C01801=1137.376,317.173,-76.633,-176.855,8.942,148.875
C01802=1137.380,316.925,-76.599,-176.858,8.938,148.874
C01803=1137.384,316.677,-76.568,-176.860,8.935,148.874
C01804=1137.388,316.429,-76.534,-176.863,8.931,148.874
C01805=1137.392,316.181,-76.503,-176.866,8.928,148.874
C01806=1137.396,315.933,-76.470,-176.869,8.923,148.874
C01807=1137.400,315.685,-76.439,-176.871,8.920,148.873
C01808=1137.405,315.438,-76.406,-176.874,8.916,148.873
C01809=1137.408,315.190,-76.374,-176.876,8.913,148.873
C01810=1137.413,314.941,-76.341,-176.879,8.909,148.873
C01811=1137.416,314.694,-76.309,-176.882,8.906,148.873
C01812=1137.420,314.447,-76.277,-176.885,8.902,148.873
C01813=1137.425,314.198,-76.245,-176.887,8.899,148.872
C01814=1137.429,313.950,-76.213,-176.890,8.894,148.872
C01815=1137.433,313.702,-76.180,-176.893,8.891,148.872
C01816=1137.437,313.424,-76.145,-176.896,8.887,148.872
C01817=1137.442,313.146,-76.109,-176.898,8.883,148.872
C01818=1137.447,312.868,-76.072,-176.901,8.879,148.871
C01819=1137.451,312.590,-76.036,-176.905,8.874,148.871
C01820=1137.456,312.342,-76.004,-176.907,8.871,148.871
C01821=1137.460,312.095,-75.973,-176.910,8.868,148.871
C01822=1137.464,311.847,-75.941,-176.913,8.864,148.870
C01823=1137.468,311.598,-75.908,-176.915,8.860,148.870
C01824=1137.472,311.350,-75.876,-176.918,8.856,148.870
C01825=1137.476,311.103,-75.845,-176.920,8.853,148.870
C01826=1137.481,310.855,-75.813,-176.924,8.849,148.870
C01827=1137.484,310.606,-75.781,-176.926,8.846,148.870
C01828=1137.489,310.359,-75.749,-176.929,8.842,148.869
C01829=1137.493,310.111,-75.717,-176.931,8.839,148.869
C01830=1137.497,309.863,-75.685,-176.934,8.835,148.869
C01831=1137.501,309.615,-75.653,-176.936,8.831,148.869
C01832=1137.505,309.367,-75.622,-176.939,8.827,148.869
C01833=1137.509,309.119,-75.589,-176.942,8.824,148.868
C01834=1137.513,308.872,-75.558,-176.945,8.820,148.868
C01835=1137.517,308.624,-75.526,-176.947,8.817,148.868
C01836=1137.521,308.376,-75.494,-176.950,8.814,148.868
C01837=1137.526,308.128,-75.462,-176.953,8.810,148.868
C01838=1137.530,307.879,-75.431,-176.955,8.806,148.868
C01839=1137.534,307.631,-75.399,-176.958,8.802,148.868
C01840=1137.538,307.384,-75.367,-176.960,8.799,148.867
C01841=1137.542,307.136,-75.336,-176.964,8.795,148.867
C01842=1137.547,306.888,-75.304,-176.966,8.792,148.867
C01843=1137.551,306.640,-75.272,-176.969,8.788,148.867
C01844=1137.554,306.392,-75.241,-176.971,8.785,148.867
C01845=1137.559,306.144,-75.209,-176.974,8.782,148.867
C01846=1137.562,305.896,-75.177,-176.977,8.777,148.866
C01847=1137.567,305.648,-75.146,-176.979,8.775,148.866
C01848=1137.571,305.400,-75.115,-176.982,8.770,148.866
C01849=1137.575,305.152,-75.082,-176.985,8.767,148.866
C01850=1137.580,304.904,-75.051,-176.988,8.763,148.866
C01851=1137.584,304.656,-75.020,-176.990,8.760,148.866
C01852=1137.588,304.409,-74.988,-176.993,8.757,148.866
C01853=1137.592,304.160,-74.957,-176.996,8.753,148.865
C01854=1137.596,303.913,-74.925,-176.998,8.750,148.865
C01855=1137.600,303.664,-74.894,-177.001,8.746,148.865
C01856=1137.604,303.417,-74.863,-177.003,8.742,148.865
C01857=1137.608,303.168,-74.831,-177.006,8.739,148.865
C01858=1137.613,302.921,-74.800,-177.009,8.735,148.865
C01859=1137.617,302.672,-74.768,-177.011,8.732,148.865
C01860=1137.621,302.425,-74.738,-177.014,8.728,148.864
C01861=1137.625,302.176,-74.706,-177.017,8.725,148.864
C01862=1137.629,301.929,-74.675,-177.019,8.722,148.864
C01863=1137.633,301.680,-74.643,-177.022,8.718,148.864
C01864=1137.638,301.433,-74.612,-177.025,8.714,148.864
C01865=1137.641,301.184,-74.581,-177.028,8.711,148.864
C01866=1137.646,300.937,-74.550,-177.030,8.707,148.864
C01867=1137.650,300.688,-74.519,-177.033,8.704,148.863
C01868=1137.654,300.441,-74.487,-177.036,8.700,148.863
C01869=1137.658,300.192,-74.456,-177.038,8.697,148.863
C01870=1137.663,299.945,-74.425,-177.041,8.693,148.863
C01871=1137.667,299.696,-74.393,-177.044,8.690,148.863
C01872=1137.671,299.448,-74.363,-177.047,8.687,148.863
C01873=1137.676,299.201,-74.331,-177.049,8.683,148.863
C01874=1137.680,298.952,-74.300,-177.052,8.680,148.863
C01875=1137.684,298.704,-74.269,-177.055,8.676,148.862
C01876=1137.687,298.456,-74.238,-177.057,8.673,148.862
C01877=1137.692,298.208,-74.207,-177.060,8.669,148.862
C01878=1137.696,297.960,-74.176,-177.063,8.665,148.862
C01879=1137.700,297.712,-74.145,-177.066,8.662,148.862
C01880=1137.705,297.464,-74.114,-177.068,8.659,148.862
C01881=1137.709,297.216,-74.083,-177.071,8.655,148.862
C01882=1137.713,296.968,-74.053,-177.074,8.652,148.862
C01883=1137.717,296.719,-74.022,-177.077,8.648,148.861
C01884=1137.721,296.471,-73.991,-177.079,8.645,148.861
C01885=1137.726,296.224,-73.959,-177.082,8.642,148.861
C01886=1137.730,295.975,-73.928,-177.085,8.638,148.861
C01887=1137.734,295.728,-73.898,-177.087,8.635,148.861
C01888=1137.738,295.480,-73.867,-177.090,8.632,148.861
C01889=1137.742,295.231,-73.836,-177.093,8.628,148.861
C01890=1137.746,294.983,-73.806,-177.095,8.624,148.861
C01891=1137.751,294.736,-73.775,-177.098,8.621,148.861
C01892=1137.755,294.487,-73.744,-177.101,8.617,148.860
C01893=1137.759,294.239,-73.713,-177.103,8.614,148.860
C01894=1137.763,293.991,-73.683,-177.106,8.610,148.860
C01895=1137.767,293.743,-73.652,-177.109,8.607,148.860
C01896=1137.772,293.495,-73.621,-177.111,8.604,148.860
C01897=1137.776,293.247,-73.591,-177.115,8.600,148.860
C01898=1137.780,292.998,-73.560,-177.117,8.597,148.860
C01899=1137.784,292.750,-73.529,-177.120,8.594,148.860
C01900=1137.788,292.503,-73.499,-177.123,8.590,148.860
C01901=1137.792,292.254,-73.468,-177.125,8.587,148.859
C01902=1137.796,292.006,-73.438,-177.128,8.584,148.859
C01903=1137.801,291.758,-73.407,-177.131,8.580,148.859
C01904=1137.805,291.511,-73.376,-177.133,8.577,148.859
C01905=1137.809,291.262,-73.346,-177.136,8.573,148.859
C01906=1137.813,291.014,-73.315,-177.139,8.569,148.859
C01907=1137.817,290.766,-73.285,-177.141,8.566,148.859
C01908=1137.822,290.518,-73.255,-177.144,8.563,148.859
C01909=1137.826,290.269,-73.223,-177.147,8.559,148.859
C01910=1137.830,290.022,-73.193,-177.150,8.556,148.859
C01911=1137.834,289.774,-73.163,-177.152,8.553,148.859
C01912=1137.839,289.525,-73.133,-177.155,8.550,148.859
C01913=1137.843,289.277,-73.102,-177.158,8.546,148.858
C01914=1137.846,289.029,-73.072,-177.160,8.543,148.858
C01915=1137.851,288.781,-73.041,-177.163,8.540,148.858
C01916=1137.855,288.533,-73.012,-177.166,8.536,148.858
C01917=1137.860,288.285,-72.981,-177.168,8.533,148.858
C01918=1137.863,288.037,-72.950,-177.171,8.530,148.858
C01919=1137.868,287.788,-72.920,-177.174,8.526,148.858
C01920=1137.873,287.513,-72.887,-177.177,8.523,148.858
C01921=1137.878,287.237,-72.853,-177.180,8.519,148.858
C01922=1137.882,286.961,-72.820,-177.183,8.515,148.858
C01923=1137.886,286.687,-72.786,-177.186,8.511,148.858
C01924=1137.891,286.438,-72.755,-177.189,8.508,148.858
C01925=1137.895,286.190,-72.726,-177.191,8.505,148.857
C01926=1137.899,285.942,-72.695,-177.195,8.501,148.857
C01927=1137.903,285.693,-72.666,-177.197,8.498,148.857
C01928=1137.907,285.446,-72.635,-177.200,8.495,148.857
C01929=1137.912,285.197,-72.605,-177.203,8.491,148.857
C01930=1137.916,284.950,-72.575,-177.206,8.488,148.857
C01931=1137.921,284.701,-72.545,-177.208,8.485,148.857
C01932=1137.924,284.453,-72.515,-177.211,8.482,148.857
C01933=1137.929,284.204,-72.485,-177.214,8.478,148.857
C01934=1137.933,283.956,-72.454,-177.216,8.475,148.857
C01935=1137.937,283.708,-72.425,-177.219,8.471,148.857
C01936=1137.941,283.461,-72.395,-177.222,8.468,148.857
C01937=1137.946,283.212,-72.365,-177.224,8.464,148.857
C01938=1137.950,282.964,-72.335,-177.227,8.461,148.857
C01939=1137.954,282.716,-72.305,-177.230,8.458,148.856
C01940=1137.958,282.468,-72.276,-177.233,8.454,148.856
C01941=1137.963,282.219,-72.246,-177.235,8.451,148.856
C01942=1137.967,281.972,-72.215,-177.238,8.448,148.856
C01943=1137.971,281.723,-72.186,-177.240,8.445,148.856
C01944=1137.976,281.475,-72.156,-177.244,8.441,148.856
C01945=1137.980,281.227,-72.126,-177.246,8.438,148.856
C01946=1137.984,280.979,-72.096,-177.249,8.435,148.856
C01947=1137.988,280.731,-72.067,-177.251,8.432,148.856
C01948=1137.993,280.482,-72.037,-177.255,8.428,148.856
C01949=1137.997,280.234,-72.007,-177.257,8.425,148.856
C01950=1138.001,279.986,-71.977,-177.260,8.422,148.856
C01951=1138.006,279.738,-71.948,-177.263,8.419,148.856
C01952=1138.010,279.489,-71.918,-177.266,8.415,148.856
C01953=1138.014,279.241,-71.889,-177.268,8.412,148.856
C01954=1138.018,278.994,-71.859,-177.271,8.409,148.856
C01955=1138.023,278.745,-71.829,-177.273,8.406,148.856
C01956=1138.027,278.497,-71.799,-177.277,8.402,148.856
C01957=1138.031,278.248,-71.770,-177.279,8.399,148.855
C01958=1138.035,278.000,-71.740,-177.282,8.396,148.856
C01959=1138.040,277.752,-71.711,-177.284,8.393,148.855
C01960=1138.044,277.504,-71.681,-177.288,8.389,148.855
C01961=1138.048,277.255,-71.652,-177.290,8.386,148.855
C01962=1138.052,277.007,-71.622,-177.293,8.383,148.855
C01963=1138.056,276.759,-71.592,-177.296,8.380,148.855
C01964=1138.060,276.511,-71.563,-177.299,8.376,148.855
C01965=1138.064,276.263,-71.533,-177.301,8.373,148.855
C01966=1138.068,276.015,-71.504,-177.304,8.370,148.855
C01967=1138.073,275.766,-71.474,-177.306,8.367,148.855
C01968=1138.077,275.518,-71.446,-177.309,8.364,148.855
C01969=1138.081,275.269,-71.416,-177.312,8.360,148.855
C01970=1138.086,275.022,-71.387,-177.315,8.357,148.855
C01971=1138.090,274.773,-71.358,-177.318,8.354,148.855
C01972=1138.094,274.525,-71.328,-177.320,8.351,148.855
C01973=1138.099,274.277,-71.299,-177.323,8.347,148.855
C01974=1138.103,274.029,-71.269,-177.326,8.344,148.855
C01975=1138.107,273.780,-71.240,-177.329,8.341,148.855
C01976=1138.111,273.532,-71.210,-177.331,8.338,148.855
C01977=1138.115,273.284,-71.181,-177.334,8.335,148.855
C01978=1138.120,273.036,-71.153,-177.337,8.331,148.855
C01979=1138.125,272.787,-71.123,-177.340,8.328,148.855
C01980=1138.129,272.539,-71.094,-177.342,8.325,148.855
C01981=1138.133,272.291,-71.064,-177.345,8.322,148.855
C01982=1138.137,272.043,-71.035,-177.348,8.319,148.855
C01983=1138.142,271.794,-71.006,-177.351,8.315,148.855
C01984=1138.146,271.546,-70.978,-177.354,8.312,148.855
C01985=1138.150,271.298,-70.948,-177.356,8.309,148.855
C01986=1138.154,271.049,-70.919,-177.359,8.306,148.855
C01987=1138.159,270.801,-70.890,-177.362,8.303,148.855
C01988=1138.163,270.553,-70.860,-177.365,8.299,148.855
C01989=1138.168,270.305,-70.831,-177.367,8.296,148.854
C01990=1138.171,270.057,-70.803,-177.370,8.293,148.855
C01991=1138.175,269.808,-70.774,-177.373,8.290,148.855
C01992=1138.180,269.559,-70.745,-177.376,8.287,148.855
C01993=1138.184,269.311,-70.716,-177.378,8.284,148.854
C01994=1138.189,269.064,-70.686,-177.381,8.280,148.855
C01995=1138.193,268.815,-70.658,-177.384,8.277,148.855
C01996=1138.197,268.567,-70.629,-177.386,8.274,148.854
C01997=1138.201,268.318,-70.600,-177.389,8.271,148.854
C01998=1138.206,268.070,-70.571,-177.392,8.268,148.855
C01999=1138.211,267.821,-70.542,-177.394,8.265,148.854
C02000=1138.214,267.573,-70.513,-177.398,8.261,148.854
C02001=1138.219,267.325,-70.485,-177.401,8.258,148.854
C02002=1138.223,267.077,-70.456,-177.403,8.255,148.855
C02003=1138.227,266.828,-70.427,-177.406,8.252,148.854
C02004=1138.231,266.580,-70.398,-177.408,8.249,148.854
C02005=1138.236,266.332,-70.370,-177.411,8.246,148.854
C02006=1138.240,266.084,-70.341,-177.414,8.242,148.854
C02007=1138.244,265.835,-70.312,-177.417,8.239,148.854
C02008=1138.249,265.588,-70.283,-177.420,8.236,148.854
C02009=1138.253,265.339,-70.255,-177.423,8.233,148.854
C02010=1138.257,265.090,-70.226,-177.425,8.230,148.854
C02011=1138.262,264.843,-70.197,-177.428,8.227,148.854
C02012=1138.266,264.594,-70.169,-177.431,8.223,148.854
C02013=1138.270,264.345,-70.140,-177.434,8.220,148.854
C02014=1138.275,264.097,-70.111,-177.436,8.217,148.854
C02015=1138.279,263.849,-70.083,-177.439,8.214,148.854
C02016=1138.283,263.600,-70.054,-177.442,8.211,148.854
C02017=1138.288,263.352,-70.026,-177.445,8.208,148.855
C02018=1138.292,263.104,-69.997,-177.447,8.205,148.854
C02019=1138.297,262.856,-69.969,-177.450,8.201,148.854
C02020=1138.301,262.607,-69.940,-177.453,8.198,148.854
C02021=1138.305,262.358,-69.912,-177.456,8.195,148.855
C02022=1138.309,262.111,-69.883,-177.458,8.192,148.854
C02023=1138.314,261.862,-69.854,-177.461,8.189,148.854
C02024=1138.318,261.589,-69.824,-177.464,8.186,148.854
C02025=1138.323,261.314,-69.792,-177.467,8.183,148.855
C02026=1138.328,261.042,-69.761,-177.471,8.179,148.855
C02027=1138.333,260.768,-69.729,-177.473,8.176,148.855
C02028=1138.337,260.519,-69.701,-177.476,8.173,148.855
C02029=1138.342,260.271,-69.673,-177.479,8.169,148.855
C02030=1138.346,260.023,-69.645,-177.482,8.166,148.855
C02031=1138.351,259.775,-69.616,-177.485,8.163,148.855
C02032=1138.354,259.526,-69.588,-177.488,8.160,148.855
C02033=1138.358,259.277,-69.560,-177.490,8.157,148.855
C02034=1138.363,259.029,-69.532,-177.493,8.154,148.855
C02035=1138.367,258.781,-69.504,-177.495,8.151,148.855
C02036=1138.372,258.532,-69.475,-177.498,8.148,148.855
C02037=1138.376,258.284,-69.447,-177.501,8.145,148.855
C02038=1138.380,258.036,-69.419,-177.504,8.142,148.855
C02039=1138.385,257.787,-69.391,-177.507,8.138,148.855
C02040=1138.389,257.539,-69.363,-177.510,8.135,148.855
C02041=1138.394,257.290,-69.334,-177.512,8.133,148.855
C02042=1138.398,257.042,-69.306,-177.515,8.130,148.855
C02043=1138.402,256.794,-69.278,-177.518,8.127,148.855
C02044=1138.407,256.546,-69.250,-177.521,8.124,148.855
C02045=1138.410,256.297,-69.222,-177.523,8.121,148.855
C02046=1138.415,256.049,-69.194,-177.526,8.118,148.855
C02047=1138.419,255.800,-69.165,-177.529,8.115,148.855
C02048=1138.424,255.552,-69.138,-177.532,8.112,148.855
C02049=1138.428,255.304,-69.110,-177.535,8.108,148.855
C02050=1138.432,255.055,-69.082,-177.538,8.105,148.855
C02051=1138.437,254.807,-69.054,-177.540,8.102,148.855
C02052=1138.441,254.559,-69.026,-177.543,8.099,148.855
C02053=1138.446,254.310,-68.999,-177.546,8.096,148.855
C02054=1138.449,254.062,-68.970,-177.548,8.093,148.855
C02055=1138.454,253.813,-68.942,-177.551,8.090,148.855
C02056=1138.458,253.565,-68.914,-177.554,8.087,148.855
C02057=1138.463,253.316,-68.887,-177.557,8.084,148.856
C02058=1138.467,253.068,-68.859,-177.559,8.081,148.855
C02059=1138.472,252.820,-68.830,-177.562,8.078,148.855
C02060=1138.476,252.571,-68.803,-177.565,8.075,148.856
C02061=1138.480,252.322,-68.775,-177.568,8.072,148.856
C02062=1138.484,252.075,-68.747,-177.571,8.069,148.856
C02063=1138.489,251.826,-68.720,-177.574,8.066,148.856
C02064=1138.493,251.577,-68.692,-177.577,8.063,148.856
C02065=1138.498,251.329,-68.664,-177.579,8.060,148.856
C02066=1138.503,251.081,-68.637,-177.582,8.057,148.856
C02067=1138.506,250.832,-68.609,-177.584,8.054,148.856
C02068=1138.511,250.584,-68.582,-177.587,8.051,148.856
C02069=1138.515,250.336,-68.554,-177.590,8.048,148.856
C02070=1138.519,250.087,-68.526,-177.593,8.045,148.856
C02071=1138.524,249.839,-68.499,-177.596,8.042,148.856
C02072=1138.528,249.590,-68.471,-177.598,8.039,148.856
C02073=1138.532,249.342,-68.443,-177.601,8.036,148.856
C02074=1138.537,249.093,-68.416,-177.604,8.033,148.856
C02075=1138.541,248.845,-68.389,-177.607,8.030,148.856
C02076=1138.546,248.596,-68.360,-177.609,8.027,148.856
C02077=1138.550,248.348,-68.333,-177.612,8.024,148.856
C02078=1138.555,248.099,-68.306,-177.615,8.021,148.856
C02079=1138.559,247.851,-68.278,-177.618,8.018,148.856
C02080=1138.563,247.602,-68.250,-177.620,8.015,148.856
C02081=1138.568,247.354,-68.223,-177.623,8.013,148.857
C02082=1138.572,247.106,-68.196,-177.627,8.009,148.857
C02083=1138.576,246.857,-68.168,-177.629,8.006,148.857
C02084=1138.581,246.608,-68.141,-177.632,8.003,148.857
C02085=1138.585,246.360,-68.113,-177.635,8.000,148.857
C02086=1138.590,246.112,-68.086,-177.638,7.997,148.857
C02087=1138.593,245.863,-68.059,-177.641,7.994,148.857
C02088=1138.598,245.615,-68.032,-177.643,7.991,148.857
C02089=1138.602,245.367,-68.005,-177.646,7.988,148.857
C02090=1138.607,245.118,-67.978,-177.648,7.985,148.857
C02091=1138.611,244.869,-67.950,-177.651,7.982,148.857
C02092=1138.615,244.621,-67.922,-177.654,7.979,148.857
C02093=1138.620,244.373,-67.895,-177.657,7.976,148.857
C02094=1138.625,244.124,-67.868,-177.660,7.974,148.857
C02095=1138.629,243.876,-67.841,-177.662,7.971,148.857
C02096=1138.633,243.626,-67.814,-177.665,7.968,148.857
C02097=1138.637,243.379,-67.787,-177.668,7.965,148.858
C02098=1138.642,243.130,-67.759,-177.671,7.962,148.858
C02099=1138.646,242.882,-67.732,-177.674,7.959,148.858
C02100=1138.651,242.633,-67.705,-177.676,7.956,148.858
C02101=1138.655,242.384,-67.678,-177.679,7.953,148.858
C02102=1138.660,242.136,-67.651,-177.682,7.950,148.858
C02103=1138.664,241.888,-67.624,-177.685,7.947,148.858
C02104=1138.668,241.639,-67.597,-177.688,7.944,148.858
C02105=1138.673,241.391,-67.570,-177.690,7.941,148.858
C02106=1138.677,241.143,-67.543,-177.693,7.939,148.858
C02107=1138.682,240.894,-67.515,-177.696,7.936,148.858
C02108=1138.685,240.645,-67.489,-177.699,7.933,148.858
C02109=1138.690,240.397,-67.462,-177.702,7.930,148.858
C02110=1138.695,240.148,-67.434,-177.704,7.927,148.859
C02111=1138.699,239.900,-67.407,-177.707,7.924,148.859
C02112=1138.703,239.652,-67.381,-177.710,7.921,148.859
C02113=1138.708,239.402,-67.355,-177.713,7.918,148.859
C02114=1138.713,239.154,-67.328,-177.716,7.915,148.859
C02115=1138.717,238.906,-67.301,-177.718,7.912,148.859
C02116=1138.721,238.657,-67.274,-177.721,7.909,148.859
C02117=1138.726,238.409,-67.247,-177.724,7.907,148.859
C02118=1138.729,238.160,-67.220,-177.727,7.904,148.859
C02119=1138.734,237.911,-67.193,-177.730,7.901,148.859
C02120=1138.739,237.663,-67.166,-177.732,7.898,148.859
C02121=1138.743,237.415,-67.140,-177.735,7.896,148.859
C02122=1138.748,237.166,-67.113,-177.738,7.893,148.860
C02123=1138.752,236.917,-67.086,-177.740,7.890,148.860
C02124=1138.756,236.669,-67.060,-177.743,7.887,148.860
C02125=1138.761,236.420,-67.033,-177.746,7.884,148.860
C02126=1138.765,236.172,-67.006,-177.749,7.881,148.860
C02127=1138.770,235.923,-66.980,-177.752,7.878,148.860
C02128=1138.775,235.652,-66.950,-177.755,7.875,148.860
C02129=1138.779,235.379,-66.921,-177.758,7.872,148.860
C02130=1138.784,235.107,-66.893,-177.761,7.869,148.860
C02131=1138.789,234.836,-66.863,-177.764,7.865,148.860
C02132=1138.794,234.587,-66.836,-177.767,7.863,148.861
C02133=1138.798,234.339,-66.810,-177.769,7.860,148.861
C02134=1138.803,234.090,-66.783,-177.772,7.857,148.861
C02135=1138.807,233.842,-66.757,-177.775,7.854,148.861
C02136=1138.812,233.593,-66.731,-177.778,7.852,148.861
C02137=1138.815,233.344,-66.704,-177.781,7.849,148.861
C02138=1138.820,233.096,-66.677,-177.783,7.846,148.861
C02139=1138.824,232.847,-66.651,-177.786,7.843,148.861
C02140=1138.829,232.599,-66.624,-177.789,7.840,148.861
C02141=1138.833,232.350,-66.599,-177.792,7.837,148.861
C02142=1138.838,232.101,-66.572,-177.795,7.834,148.861
C02143=1138.842,231.853,-66.546,-177.797,7.831,148.862
C02144=1138.847,231.604,-66.519,-177.800,7.828,148.862
C02145=1138.851,231.356,-66.492,-177.803,7.826,148.862
C02146=1138.855,231.107,-66.466,-177.806,7.823,148.862
C02147=1138.860,230.858,-66.440,-177.808,7.821,148.862
C02148=1138.864,230.611,-66.414,-177.811,7.818,148.862
C02149=1138.869,230.361,-66.388,-177.814,7.815,148.862
C02150=1138.873,230.113,-66.361,-177.817,7.812,148.862
C02151=1138.878,229.864,-66.335,-177.820,7.809,148.862
C02152=1138.882,229.616,-66.308,-177.822,7.806,148.863
C02153=1138.886,229.367,-66.283,-177.825,7.803,148.863
C02154=1138.891,229.119,-66.256,-177.828,7.800,148.863
C02155=1138.895,228.870,-66.230,-177.831,7.797,148.863
C02156=1138.900,228.622,-66.204,-177.834,7.795,148.863
C02157=1138.905,228.373,-66.177,-177.837,7.792,148.863
C02158=1138.909,228.124,-66.152,-177.840,7.789,148.863
C02159=1138.913,227.876,-66.126,-177.842,7.787,148.863
C02160=1138.917,227.627,-66.099,-177.845,7.784,148.864
C02161=1138.922,227.378,-66.073,-177.848,7.781,148.864
C02162=1138.926,227.129,-66.047,-177.850,7.778,148.864
C02163=1138.931,226.881,-66.022,-177.853,7.775,148.864
C02164=1138.936,226.633,-65.995,-177.856,7.772,148.864
C02165=1138.940,226.384,-65.969,-177.859,7.770,148.864
C02166=1138.944,226.135,-65.943,-177.862,7.767,148.864
C02167=1138.948,225.886,-65.918,-177.865,7.764,148.864
C02168=1138.954,225.639,-65.891,-177.867,7.762,148.864
C02169=1138.958,225.390,-65.865,-177.870,7.759,148.865
C02170=1138.962,225.141,-65.839,-177.873,7.756,148.865
C02171=1138.966,224.892,-65.814,-177.876,7.753,148.865
C02172=1138.971,224.643,-65.788,-177.879,7.751,148.865
C02173=1138.976,224.395,-65.762,-177.882,7.748,148.865
C02174=1138.980,224.147,-65.735,-177.884,7.745,148.865
C02175=1138.984,223.898,-65.710,-177.887,7.742,148.865
C02176=1138.989,223.649,-65.684,-177.889,7.740,148.865
C02177=1138.993,223.401,-65.659,-177.892,7.737,148.866
C02178=1138.998,223.152,-65.633,-177.895,7.734,148.866
C02179=1139.003,222.903,-65.607,-177.898,7.731,148.866
C02180=1139.007,222.654,-65.581,-177.901,7.729,148.866
C02181=1139.012,222.406,-65.555,-177.904,7.726,148.866
C02182=1139.016,222.158,-65.530,-177.907,7.723,148.866
C02183=1139.020,221.909,-65.504,-177.909,7.721,148.866
C02184=1139.025,221.661,-65.478,-177.912,7.718,148.866
C02185=1139.029,221.412,-65.453,-177.915,7.715,148.867
C02186=1139.033,221.163,-65.427,-177.918,7.712,148.867
C02187=1139.038,220.914,-65.401,-177.921,7.709,148.867
C02188=1139.042,220.666,-65.376,-177.923,7.706,148.867
C02189=1139.047,220.417,-65.350,-177.926,7.704,148.867
C02190=1139.051,220.168,-65.324,-177.929,7.702,148.867
C02191=1139.056,219.920,-65.298,-177.932,7.699,148.868
C02192=1139.061,219.671,-65.273,-177.935,7.696,148.868
C02193=1139.065,219.422,-65.248,-177.937,7.693,148.868
C02194=1139.070,219.174,-65.222,-177.940,7.690,148.868
C02195=1139.074,218.925,-65.196,-177.943,7.688,148.868
C02196=1139.078,218.676,-65.171,-177.946,7.686,148.868
C02197=1139.083,218.428,-65.146,-177.948,7.683,148.868
C02198=1139.087,218.179,-65.121,-177.951,7.680,148.868
C02199=1139.091,217.930,-65.095,-177.954,7.677,148.869
C02200=1139.096,217.682,-65.070,-177.957,7.674,148.869
C02201=1139.100,217.433,-65.044,-177.960,7.671,148.869
C02202=1139.105,217.185,-65.019,-177.962,7.669,148.869
C02203=1139.110,216.936,-64.994,-177.965,7.666,148.869
C02204=1139.114,216.687,-64.968,-177.968,7.663,148.869
C02205=1139.119,216.439,-64.942,-177.971,7.661,148.870
C02206=1139.123,216.189,-64.917,-177.974,7.658,148.870
C02207=1139.128,215.941,-64.892,-177.976,7.656,148.870
C02208=1139.132,215.692,-64.866,-177.979,7.653,148.870
C02209=1139.136,215.443,-64.842,-177.982,7.650,148.870
C02210=1139.141,215.195,-64.816,-177.985,7.648,148.870
C02211=1139.145,214.946,-64.791,-177.988,7.645,148.870
C02212=1139.150,214.698,-64.766,-177.990,7.643,148.871
C02213=1139.155,214.449,-64.740,-177.993,7.640,148.871
C02214=1139.159,214.201,-64.715,-177.996,7.637,148.871
C02215=1139.164,213.951,-64.690,-177.999,7.634,148.871
C02216=1139.168,213.704,-64.665,-178.002,7.631,148.871
C02217=1139.173,213.454,-64.640,-178.005,7.630,148.872
C02218=1139.177,213.205,-64.614,-178.007,7.627,148.872
C02219=1139.182,212.957,-64.590,-178.010,7.624,148.872
C02220=1139.185,212.708,-64.564,-178.013,7.621,148.872
C02221=1139.190,212.459,-64.540,-178.016,7.618,148.872
C02222=1139.195,212.211,-64.514,-178.018,7.616,148.872
C02223=1139.200,211.962,-64.489,-178.021,7.613,148.872
C02224=1139.204,211.713,-64.464,-178.025,7.611,148.873
C02225=1139.208,211.465,-64.440,-178.027,7.608,148.873
C02226=1139.213,211.216,-64.414,-178.030,7.606,148.873
C02227=1139.218,210.967,-64.389,-178.032,7.603,148.873
C02228=1139.221,210.719,-64.364,-178.036,7.600,148.873
C02229=1139.226,210.470,-64.339,-178.038,7.597,148.873
C02230=1139.232,210.221,-64.315,-178.041,7.594,148.874
C02231=1139.236,209.972,-64.289,-178.044,7.593,148.874
C02232=1139.240,209.701,-64.262,-178.047,7.590,148.874
C02233=1139.245,209.431,-64.235,-178.050,7.587,148.874
C02234=1139.250,209.160,-64.208,-178.053,7.584,148.874
C02235=1139.255,208.890,-64.181,-178.056,7.581,148.875
C02236=1139.260,208.641,-64.156,-178.058,7.579,148.875
C02237=1139.265,208.392,-64.132,-178.062,7.576,148.875
C02238=1139.268,208.144,-64.106,-178.065,7.573,148.875
C02239=1139.273,207.895,-64.082,-178.067,7.570,148.875
C02240=1139.278,207.646,-64.058,-178.070,7.568,148.876
C02241=1139.282,207.397,-64.033,-178.073,7.566,148.876
C02242=1139.287,207.149,-64.007,-178.076,7.563,148.876
C02243=1139.291,206.900,-63.983,-178.079,7.560,148.876
C02244=1139.296,206.651,-63.958,-178.081,7.558,148.876
C02245=1139.301,206.403,-63.934,-178.084,7.555,148.876
C02246=1139.305,206.153,-63.909,-178.087,7.553,148.877
C02247=1139.309,205.905,-63.884,-178.090,7.550,148.877
C02248=1139.314,205.657,-63.860,-178.092,7.548,148.877
C02249=1139.319,205.407,-63.835,-178.096,7.545,148.877
C02250=1139.323,205.159,-63.810,-178.098,7.542,148.877
C02251=1139.328,204.910,-63.786,-178.101,7.540,148.877
C02252=1139.332,204.661,-63.761,-178.104,7.537,148.878
C02253=1139.337,204.412,-63.737,-178.107,7.535,148.878
C02254=1139.342,204.164,-63.713,-178.110,7.532,148.878
C02255=1139.346,203.915,-63.688,-178.112,7.530,148.878
C02256=1139.351,203.666,-63.663,-178.115,7.527,148.878
C02257=1139.355,203.418,-63.639,-178.118,7.524,148.879
C02258=1139.360,203.168,-63.614,-178.120,7.522,148.879
C02259=1139.364,202.920,-63.590,-178.123,7.519,148.879
C02260=1139.369,202.671,-63.566,-178.127,7.517,148.879
C02261=1139.373,202.422,-63.541,-178.129,7.514,148.879
C02262=1139.378,202.173,-63.517,-178.132,7.512,148.880
C02263=1139.382,201.925,-63.492,-178.135,7.509,148.880
C02264=1139.387,201.676,-63.468,-178.138,7.506,148.880
C02265=1139.391,201.427,-63.443,-178.140,7.505,148.880
C02266=1139.396,201.179,-63.419,-178.143,7.502,148.880
C02267=1139.401,200.930,-63.395,-178.146,7.499,148.881
C02268=1139.405,200.681,-63.370,-178.149,7.497,148.881
C02269=1139.409,200.432,-63.346,-178.151,7.494,148.881
C02270=1139.414,200.184,-63.321,-178.155,7.492,148.881
C02271=1139.419,199.935,-63.297,-178.157,7.490,148.881
C02272=1139.423,199.686,-63.274,-178.160,7.487,148.882
C02273=1139.428,199.437,-63.249,-178.163,7.484,148.882
C02274=1139.432,199.188,-63.225,-178.165,7.482,148.882
C02275=1139.437,198.940,-63.201,-178.169,7.480,148.882
C02276=1139.441,198.692,-63.177,-178.171,7.477,148.882
C02277=1139.446,198.442,-63.152,-178.174,7.474,148.883
C02278=1139.450,198.193,-63.128,-178.177,7.472,148.883
C02279=1139.455,197.945,-63.104,-178.180,7.469,148.883
C02280=1139.460,197.696,-63.080,-178.183,7.467,148.883
C02281=1139.464,197.447,-63.056,-178.185,7.465,148.884
C02282=1139.468,197.198,-63.032,-178.188,7.462,148.884
C02283=1139.473,196.949,-63.008,-178.191,7.460,148.884
C02284=1139.478,196.700,-62.984,-178.194,7.457,148.884
C02285=1139.482,196.452,-62.960,-178.197,7.454,148.884
C02286=1139.487,196.203,-62.936,-178.199,7.452,148.885
C02287=1139.492,195.954,-62.912,-178.202,7.450,148.885
C02288=1139.495,195.705,-62.888,-178.205,7.447,148.885
C02289=1139.500,195.456,-62.863,-178.208,7.445,148.885
C02290=1139.505,195.207,-62.840,-178.211,7.442,148.885
C02291=1139.510,194.959,-62.816,-178.213,7.439,148.886
C02292=1139.514,194.710,-62.792,-178.216,7.438,148.886
C02293=1139.519,194.461,-62.768,-178.219,7.435,148.886
C02294=1139.523,194.213,-62.744,-178.222,7.432,148.886
C02295=1139.528,193.964,-62.720,-178.224,7.430,148.887
C02296=1139.532,193.715,-62.696,-178.228,7.428,148.887
C02297=1139.537,193.466,-62.672,-178.230,7.425,148.887
C02298=1139.541,193.217,-62.648,-178.233,7.423,148.887
C02299=1139.546,192.968,-62.625,-178.236,7.420,148.887
C02300=1139.550,192.720,-62.601,-178.239,7.418,148.888
C02301=1139.555,192.471,-62.578,-178.242,7.415,148.888
C02302=1139.560,192.222,-62.554,-178.245,7.413,148.888
C02303=1139.564,191.973,-62.530,-178.247,7.411,148.888
C02304=1139.569,191.724,-62.507,-178.250,7.408,148.889
C02305=1139.573,191.476,-62.483,-178.253,7.406,148.889
C02306=1139.579,191.226,-62.459,-178.256,7.404,148.889
C02307=1139.583,190.978,-62.435,-178.259,7.401,148.889
C02308=1139.588,190.729,-62.411,-178.261,7.399,148.889
C02309=1139.593,190.480,-62.388,-178.264,7.396,148.890
C02310=1139.597,190.232,-62.364,-178.266,7.394,148.890
C02311=1139.602,189.983,-62.341,-178.270,7.391,148.890
C02312=1139.606,189.734,-62.317,-178.272,7.389,148.890
C02313=1139.610,189.484,-62.293,-178.275,7.387,148.891
C02314=1139.615,189.235,-62.269,-178.278,7.384,148.891
C02315=1139.620,188.986,-62.246,-178.281,7.382,148.891
C02316=1139.624,188.738,-62.222,-178.284,7.380,148.892
C02317=1139.629,188.490,-62.199,-178.287,7.377,148.892
C02318=1139.633,188.241,-62.176,-178.289,7.375,148.892
C02319=1139.638,187.992,-62.153,-178.292,7.372,148.892
C02320=1139.642,187.743,-62.129,-178.295,7.370,148.893
C02321=1139.647,187.494,-62.105,-178.298,7.368,148.893
C02322=1139.652,187.245,-62.082,-178.301,7.365,148.893
C02323=1139.656,186.996,-62.059,-178.303,7.363,148.893
C02324=1139.661,186.747,-62.035,-178.307,7.360,148.893
C02325=1139.666,186.498,-62.012,-178.309,7.358,148.894
C02326=1139.670,186.250,-61.988,-178.312,7.356,148.894
C02327=1139.675,186.001,-61.965,-178.314,7.354,148.894
C02328=1139.679,185.752,-61.942,-178.318,7.351,148.894
C02329=1139.684,185.503,-61.918,-178.320,7.348,148.895
C02330=1139.688,185.254,-61.895,-178.323,7.346,148.895
C02331=1139.693,185.005,-61.872,-178.326,7.344,148.895
C02332=1139.698,184.756,-61.848,-178.329,7.342,148.895
C02333=1139.702,184.507,-61.825,-178.332,7.339,148.896
C02334=1139.706,184.258,-61.802,-178.334,7.337,148.896
C02335=1139.712,184.010,-61.779,-178.337,7.335,148.896
C02336=1139.716,183.740,-61.753,-178.340,7.332,148.896
C02337=1139.721,183.470,-61.728,-178.344,7.329,148.897
C02338=1139.727,183.200,-61.703,-178.346,7.328,148.897
C02339=1139.731,182.931,-61.679,-178.349,7.325,148.897
C02340=1139.736,182.682,-61.655,-178.352,7.322,148.897
C02341=1139.741,182.433,-61.632,-178.355,7.320,148.898
C02342=1139.745,182.184,-61.609,-178.358,7.317,148.898
C02343=1139.749,181.935,-61.586,-178.361,7.316,148.898
C02344=1139.755,181.687,-61.563,-178.363,7.313,148.898
C02345=1139.759,181.438,-61.539,-178.367,7.310,148.899
C02346=1139.763,181.189,-61.517,-178.369,7.308,148.899
C02347=1139.768,180.940,-61.493,-178.372,7.306,148.899
C02348=1139.773,180.691,-61.470,-178.375,7.304,148.900
C02349=1139.777,180.442,-61.447,-178.378,7.301,148.900
C02350=1139.782,180.193,-61.425,-178.380,7.299,148.900
C02351=1139.787,179.944,-61.402,-178.383,7.296,148.900
C02352=1139.791,179.696,-61.379,-178.386,7.295,148.901
C02353=1139.796,179.447,-61.355,-178.389,7.292,148.901
C02354=1139.800,179.198,-61.332,-178.391,7.290,148.901
C02355=1139.805,178.949,-61.310,-178.395,7.288,148.901
C02356=1139.810,178.700,-61.287,-178.397,7.285,148.902
C02357=1139.815,178.451,-61.264,-178.400,7.283,148.902
C02358=1139.819,178.202,-61.241,-178.403,7.281,148.902
C02359=1139.824,177.952,-61.218,-178.406,7.278,148.902
C02360=1139.828,177.704,-61.196,-178.408,7.277,148.903
C02361=1139.833,177.455,-61.172,-178.411,7.274,148.903
C02362=1139.837,177.206,-61.149,-178.414,7.272,148.903
C02363=1139.842,176.957,-61.127,-178.417,7.269,148.904
C02364=1139.847,176.709,-61.104,-178.420,7.267,148.904
C02365=1139.851,176.460,-61.081,-178.423,7.265,148.904
C02366=1139.856,176.210,-61.059,-178.425,7.263,148.904
C02367=1139.860,175.962,-61.036,-178.428,7.260,148.905
C02368=1139.865,175.713,-61.013,-178.431,7.259,148.905
C02369=1139.870,175.464,-60.991,-178.434,7.256,148.905
C02370=1139.874,175.215,-60.967,-178.437,7.254,148.906
C02371=1139.879,174.966,-60.946,-178.440,7.251,148.906
C02372=1139.884,174.717,-60.922,-178.442,7.249,148.906
C02373=1139.888,174.468,-60.900,-178.445,7.247,148.906
C02374=1139.893,174.219,-60.877,-178.448,7.245,148.907
C02375=1139.897,173.971,-60.855,-178.451,7.242,148.907
C02376=1139.902,173.721,-60.832,-178.454,7.240,148.907
C02377=1139.906,173.473,-60.809,-178.456,7.238,148.907
C02378=1139.912,173.224,-60.787,-178.459,7.236,148.908
C02379=1139.916,172.975,-60.764,-178.462,7.234,148.908
C02380=1139.920,172.725,-60.742,-178.465,7.231,148.908
C02381=1139.926,172.477,-60.720,-178.467,7.229,148.909
C02382=1139.930,172.228,-60.697,-178.471,7.227,148.909
C02383=1139.935,171.978,-60.674,-178.473,7.225,148.909
C02384=1139.939,171.730,-60.652,-178.476,7.222,148.909
C02385=1139.944,171.480,-60.629,-178.479,7.221,148.910
C02386=1139.949,171.232,-60.607,-178.482,7.218,148.910
C02387=1139.953,170.983,-60.585,-178.484,7.216,148.910
C02388=1139.958,170.733,-60.562,-178.488,7.213,148.911
C02389=1139.963,170.485,-60.540,-178.490,7.211,148.911
C02390=1139.967,170.236,-60.518,-178.493,7.210,148.911
C02391=1139.973,169.987,-60.496,-178.496,7.207,148.912
C02392=1139.977,169.738,-60.473,-178.498,7.205,148.912
C02393=1139.981,169.489,-60.451,-178.501,7.203,148.912
C02394=1139.986,169.240,-60.429,-178.504,7.201,148.912
C02395=1139.990,168.991,-60.406,-178.507,7.198,148.913
C02396=1139.995,168.743,-60.384,-178.510,7.196,148.913
C02397=1140.000,168.493,-60.361,-178.513,7.194,148.913
C02398=1140.005,168.244,-60.339,-178.516,7.192,148.914
C02399=1140.009,167.996,-60.317,-178.518,7.190,148.914
C02400=1140.013,167.746,-60.295,-178.521,7.187,148.914
C02401=1140.019,167.497,-60.273,-178.524,7.186,148.915
C02402=1140.023,167.248,-60.251,-178.527,7.183,148.915
C02403=1140.028,167.000,-60.228,-178.529,7.181,148.915
C02404=1140.032,166.751,-60.206,-178.532,7.179,148.915
C02405=1140.038,166.502,-60.184,-178.535,7.177,148.916
C02406=1140.042,166.252,-60.162,-178.538,7.175,148.916
C02407=1140.047,166.004,-60.140,-178.541,7.172,148.916
C02408=1140.051,165.755,-60.118,-178.544,7.170,148.917
C02409=1140.056,165.506,-60.096,-178.546,7.168,148.917
C02410=1140.061,165.257,-60.073,-178.549,7.166,148.917
C02411=1140.066,165.008,-60.051,-178.552,7.164,148.918
C02412=1140.070,164.759,-60.029,-178.555,7.162,148.918
C02413=1140.075,164.510,-60.008,-178.557,7.160,148.918
C02414=1140.079,164.261,-59.986,-178.561,7.157,148.918
C02415=1140.084,164.012,-59.964,-178.563,7.155,148.919
C02416=1140.088,163.763,-59.942,-178.566,7.153,148.919
C02417=1140.094,163.514,-59.920,-178.569,7.151,148.919
C02418=1140.098,163.265,-59.898,-178.572,7.149,148.920
C02419=1140.103,163.016,-59.876,-178.574,7.147,148.920
C02420=1140.107,162.767,-59.854,-178.577,7.144,148.920
C02421=1140.112,162.518,-59.832,-178.580,7.143,148.921
C02422=1140.116,162.269,-59.810,-178.583,7.140,148.921
C02423=1140.121,162.020,-59.788,-178.586,7.138,148.921
C02424=1140.126,161.771,-59.767,-178.588,7.136,148.921
C02425=1140.130,161.522,-59.745,-178.591,7.134,148.922
C02426=1140.135,161.273,-59.723,-178.594,7.132,148.922
C02427=1140.139,161.024,-59.701,-178.597,7.130,148.923
C02428=1140.144,160.775,-59.679,-178.600,7.127,148.923
C02429=1140.149,160.525,-59.658,-178.602,7.126,148.923
C02430=1140.154,160.277,-59.636,-178.606,7.123,148.923
C02431=1140.159,160.028,-59.615,-178.608,7.122,148.924
C02432=1140.163,159.779,-59.593,-178.611,7.119,148.924
C02433=1140.168,159.530,-59.571,-178.614,7.117,148.924
C02434=1140.172,159.281,-59.549,-178.617,7.115,148.925
C02435=1140.177,159.032,-59.528,-178.619,7.113,148.925
C02436=1140.182,158.783,-59.506,-178.623,7.111,148.925
C02437=1140.186,158.534,-59.484,-178.625,7.109,148.926
C02438=1140.191,158.285,-59.462,-178.628,7.107,148.926
C02439=1140.196,158.036,-59.441,-178.631,7.105,148.926
C02440=1140.201,157.767,-59.417,-178.634,7.103,148.927
C02441=1140.206,157.498,-59.395,-178.637,7.100,148.927
C02442=1140.211,157.229,-59.371,-178.640,7.098,148.927
C02443=1140.216,156.960,-59.348,-178.643,7.096,148.928
C02444=1140.221,156.711,-59.326,-178.646,7.093,148.928
C02445=1140.226,156.462,-59.305,-178.648,7.092,148.928
C02446=1140.230,156.213,-59.283,-178.651,7.090,148.929
C02447=1140.235,155.964,-59.261,-178.654,7.088,148.929
C02448=1140.240,155.714,-59.240,-178.657,7.086,148.929
C02449=1140.245,155.466,-59.218,-178.659,7.084,148.930
C02450=1140.249,155.217,-59.198,-178.662,7.082,148.930
C02451=1140.253,154.967,-59.176,-178.665,7.079,148.930
C02452=1140.258,154.719,-59.154,-178.668,7.078,148.931
C02453=1140.264,154.469,-59.133,-178.671,7.076,148.931
C02454=1140.268,154.221,-59.112,-178.674,7.073,148.931
C02455=1140.273,153.971,-59.090,-178.676,7.071,148.932
C02456=1140.277,153.723,-59.069,-178.679,7.070,148.932
C02457=1140.282,153.473,-59.048,-178.682,7.067,148.932
C02458=1140.287,153.225,-59.027,-178.685,7.065,148.933
C02459=1140.291,152.975,-59.004,-178.687,7.063,148.933
C02460=1140.297,152.726,-58.984,-178.691,7.061,148.933
C02461=1140.301,152.478,-58.962,-178.693,7.059,148.934
C02462=1140.306,152.228,-58.941,-178.696,7.057,148.934
C02463=1140.310,151.978,-58.920,-178.699,7.056,148.934
C02464=1140.315,151.730,-58.898,-178.702,7.053,148.935
C02465=1140.320,151.481,-58.878,-178.704,7.051,148.935
C02466=1140.325,151.232,-58.856,-178.707,7.049,148.935
C02467=1140.329,150.982,-58.835,-178.710,7.047,148.936
C02468=1140.334,150.734,-58.813,-178.713,7.045,148.936
C02469=1140.339,150.485,-58.793,-178.716,7.043,148.937
C02470=1140.344,150.235,-58.772,-178.719,7.041,148.937
C02471=1140.349,149.987,-58.750,-178.721,7.039,148.937
C02472=1140.353,149.738,-58.730,-178.724,7.037,148.937
C02473=1140.357,149.488,-58.708,-178.727,7.035,148.938
C02474=1140.362,149.239,-58.687,-178.730,7.033,148.938
C02475=1140.367,148.990,-58.667,-178.733,7.031,148.939
C02476=1140.372,148.741,-58.646,-178.735,7.029,148.939
C02477=1140.377,148.492,-58.624,-178.738,7.027,148.939
C02478=1140.381,148.243,-58.604,-178.741,7.025,148.939
C02479=1140.386,147.993,-58.582,-178.744,7.023,148.940
C02480=1140.391,147.745,-58.561,-178.746,7.021,148.940
C02481=1140.395,147.496,-58.540,-178.750,7.019,148.941
C02482=1140.400,147.247,-58.519,-178.752,7.017,148.941
C02483=1140.405,146.998,-58.499,-178.755,7.016,148.941
C02484=1140.410,146.749,-58.477,-178.757,7.013,148.942
C02485=1140.415,146.500,-58.456,-178.761,7.011,148.942
C02486=1140.419,146.251,-58.436,-178.763,7.009,148.942
C02487=1140.424,146.001,-58.415,-178.766,7.008,148.943
C02488=1140.428,145.752,-58.394,-178.769,7.006,148.943
C02489=1140.433,145.503,-58.372,-178.772,7.003,148.943
C02490=1140.438,145.254,-58.352,-178.775,7.002,148.944
C02491=1140.443,145.005,-58.331,-178.778,7.000,148.944
C02492=1140.447,144.756,-58.311,-178.780,6.998,148.944
C02493=1140.452,144.507,-58.290,-178.783,6.995,148.945
C02494=1140.457,144.258,-58.269,-178.786,6.994,148.945
C02495=1140.462,144.009,-58.248,-178.788,6.992,148.946
C02496=1140.466,143.760,-58.228,-178.791,6.990,148.946
C02497=1140.472,143.510,-58.207,-178.794,6.989,148.946
C02498=1140.476,143.262,-58.187,-178.797,6.986,148.947
C02499=1140.481,143.013,-58.165,-178.800,6.984,148.947
C02500=1140.485,142.763,-58.144,-178.803,6.983,148.947
C02501=1140.490,142.514,-58.123,-178.805,6.981,148.948
C02502=1140.494,142.265,-58.103,-178.808,6.978,148.948
C02503=1140.500,142.016,-58.082,-178.811,6.976,148.948
C02504=1140.504,141.767,-58.062,-178.814,6.975,148.949
C02505=1140.508,141.518,-58.041,-178.816,6.973,148.949
C02506=1140.514,141.269,-58.020,-178.819,6.971,148.950
C02507=1140.518,141.019,-58.001,-178.822,6.969,148.950
C02508=1140.524,140.770,-57.980,-178.825,6.967,148.950
C02509=1140.528,140.521,-57.959,-178.828,6.965,148.951
C02510=1140.532,140.272,-57.939,-178.831,6.964,148.951
C02511=1140.538,140.023,-57.918,-178.833,6.961,148.951
C02512=1140.542,139.774,-57.898,-178.836,6.959,148.952
C02513=1140.546,139.525,-57.877,-178.839,6.957,148.952
C02514=1140.552,139.275,-57.856,-178.842,6.956,148.952
C02515=1140.556,139.026,-57.836,-178.844,6.954,148.953
C02516=1140.561,138.778,-57.816,-178.847,6.952,148.953
C02517=1140.566,138.528,-57.795,-178.850,6.950,148.954
C02518=1140.571,138.279,-57.775,-178.853,6.948,148.954
C02519=1140.575,138.030,-57.755,-178.856,6.946,148.954
C02520=1140.581,137.781,-57.734,-178.858,6.945,148.955
C02521=1140.585,137.532,-57.714,-178.861,6.943,148.955
C02522=1140.590,137.283,-57.694,-178.864,6.940,148.956
C02523=1140.594,137.034,-57.674,-178.867,6.939,148.956
C02524=1140.599,136.784,-57.653,-178.869,6.937,148.956
C02525=1140.604,136.536,-57.632,-178.872,6.935,148.957
C02526=1140.609,136.286,-57.613,-178.875,6.933,148.957
C02527=1140.613,136.037,-57.592,-178.878,6.931,148.957
C02528=1140.618,135.788,-57.571,-178.881,6.929,148.958
C02529=1140.623,135.539,-57.551,-178.884,6.927,148.958
C02530=1140.628,135.290,-57.532,-178.886,6.926,148.958
C02531=1140.632,135.041,-57.511,-178.889,6.924,148.959
C02532=1140.638,134.792,-57.490,-178.892,6.922,148.959
C02533=1140.642,134.542,-57.471,-178.894,6.920,148.960
C02534=1140.647,134.293,-57.450,-178.898,6.918,148.960
C02535=1140.652,134.044,-57.430,-178.900,6.916,148.960
C02536=1140.656,133.795,-57.410,-178.903,6.915,148.961
C02537=1140.661,133.545,-57.389,-178.906,6.913,148.961
C02538=1140.667,133.297,-57.370,-178.909,6.911,148.962
C02539=1140.671,133.048,-57.349,-178.911,6.909,148.962
C02540=1140.676,132.798,-57.330,-178.914,6.908,148.962
C02541=1140.680,132.549,-57.309,-178.917,6.905,148.963
C02542=1140.685,132.300,-57.289,-178.920,6.904,148.963
C02543=1140.689,132.051,-57.269,-178.923,6.902,148.964
C02544=1140.695,131.782,-57.248,-178.926,6.900,148.964
C02545=1140.700,131.514,-57.226,-178.929,6.898,148.964
C02546=1140.706,131.245,-57.205,-178.932,6.896,148.965
C02547=1140.711,130.977,-57.184,-178.934,6.894,148.965
C02548=1140.715,130.728,-57.163,-178.938,6.892,148.966
C02549=1140.720,130.478,-57.144,-178.940,6.890,148.966
C02550=1140.724,130.229,-57.123,-178.943,6.888,148.966
C02551=1140.729,129.980,-57.103,-178.946,6.887,148.967
C02552=1140.735,129.731,-57.083,-178.949,6.885,148.967
C02553=1140.740,129.482,-57.063,-178.951,6.883,148.967
C02554=1140.744,129.233,-57.043,-178.954,6.882,148.968
C02555=1140.749,128.983,-57.023,-178.957,6.880,148.968
C02556=1140.754,128.734,-57.004,-178.960,6.877,148.969
C02557=1140.759,128.485,-56.984,-178.963,6.876,148.969
C02558=1140.763,128.236,-56.964,-178.965,6.874,148.969
C02559=1140.768,127.986,-56.944,-178.968,6.872,148.970
C02560=1140.773,127.738,-56.924,-178.971,6.871,148.970
C02561=1140.778,127.488,-56.905,-178.974,6.869,148.971
C02562=1140.783,127.239,-56.885,-178.976,6.867,148.971
C02563=1140.787,126.990,-56.865,-178.979,6.866,148.971
C02564=1140.792,126.741,-56.845,-178.982,6.864,148.972
C02565=1140.796,126.492,-56.826,-178.984,6.862,148.972
C02566=1140.801,126.243,-56.806,-178.988,6.860,148.973
C02567=1140.806,125.994,-56.787,-178.991,6.858,148.973
C02568=1140.811,125.744,-56.767,-178.993,6.856,148.973
C02569=1140.816,125.495,-56.747,-178.996,6.855,148.974
C02570=1140.820,125.246,-56.727,-178.999,6.853,148.974
C02571=1140.825,124.997,-56.708,-179.001,6.851,148.975
C02572=1140.830,124.747,-56.688,-179.004,6.849,148.975
C02573=1140.835,124.498,-56.668,-179.007,6.848,148.975
C02574=1140.840,124.249,-56.649,-179.010,6.846,148.976
C02575=1140.844,124.000,-56.630,-179.012,6.844,148.976
C02576=1140.849,123.751,-56.610,-179.015,6.843,148.977
C02577=1140.854,123.502,-56.590,-179.018,6.841,148.977
C02578=1140.859,123.252,-56.571,-179.021,6.838,148.977
C02579=1140.864,123.003,-56.551,-179.024,6.837,148.978
C02580=1140.869,122.754,-56.532,-179.027,6.835,148.978
C02581=1140.874,122.504,-56.512,-179.029,6.833,148.979
C02582=1140.878,122.256,-56.493,-179.032,6.832,148.979
C02583=1140.883,122.006,-56.474,-179.035,6.830,148.979
C02584=1140.887,121.757,-56.453,-179.037,6.828,148.980
C02585=1140.893,121.508,-56.434,-179.040,6.827,148.980
C02586=1140.897,121.259,-56.414,-179.043,6.825,148.981
C02587=1140.902,121.010,-56.396,-179.046,6.823,148.981
C02588=1140.907,120.761,-56.376,-179.048,6.822,148.981
C02589=1140.912,120.511,-56.356,-179.051,6.820,148.982
C02590=1140.917,120.262,-56.337,-179.054,6.818,148.982
C02591=1140.921,120.013,-56.318,-179.057,6.817,148.983
C02592=1140.926,119.764,-56.299,-179.060,6.815,148.983
C02593=1140.931,119.514,-56.279,-179.062,6.813,148.984
C02594=1140.936,119.265,-56.259,-179.065,6.812,148.984
C02595=1140.940,119.016,-56.241,-179.068,6.810,148.984
C02596=1140.945,118.767,-56.221,-179.071,6.808,148.985
C02597=1140.951,118.517,-56.202,-179.074,6.806,148.985
C02598=1140.955,118.268,-56.183,-179.077,6.804,148.986
C02599=1140.960,118.019,-56.164,-179.079,6.803,148.986
C02600=1140.965,117.770,-56.144,-179.082,6.801,148.987
C02601=1140.969,117.521,-56.126,-179.085,6.799,148.987
C02602=1140.974,117.271,-56.106,-179.088,6.797,148.987
C02603=1140.980,117.023,-56.087,-179.090,6.796,148.988
C02604=1140.984,116.773,-56.068,-179.093,6.794,148.988
C02605=1140.989,116.523,-56.049,-179.096,6.792,148.989
C02606=1140.994,116.274,-56.029,-179.098,6.791,148.989
C02607=1140.998,116.025,-56.010,-179.101,6.789,148.989
C02608=1141.003,115.776,-55.991,-179.104,6.787,148.990
C02609=1141.008,115.527,-55.971,-179.107,6.786,148.990
C02610=1141.013,115.277,-55.953,-179.110,6.784,148.991
C02611=1141.018,115.029,-55.934,-179.113,6.783,148.991
C02612=1141.022,114.779,-55.915,-179.115,6.781,148.992
C02613=1141.028,114.530,-55.896,-179.118,6.779,148.992
C02614=1141.033,114.280,-55.877,-179.121,6.778,148.992
C02615=1141.037,114.032,-55.858,-179.124,6.776,148.993
C02616=1141.042,113.782,-55.839,-179.126,6.774,148.993
C02617=1141.047,113.534,-55.820,-179.129,6.773,148.994
C02618=1141.052,113.283,-55.801,-179.132,6.771,148.994
C02619=1141.056,113.035,-55.782,-179.134,6.769,148.994
C02620=1141.061,112.785,-55.763,-179.137,6.767,148.995
C02621=1141.066,112.536,-55.745,-179.140,6.766,148.995
C02622=1141.071,112.287,-55.725,-179.143,6.764,148.996
C02623=1141.075,112.038,-55.706,-179.146,6.763,148.996
C02624=1141.081,111.788,-55.688,-179.149,6.761,148.997
C02625=1141.085,111.539,-55.669,-179.151,6.759,148.997
C02626=1141.091,111.290,-55.650,-179.154,6.758,148.998
C02627=1141.095,111.041,-55.631,-179.157,6.756,148.998
C02628=1141.100,110.792,-55.612,-179.159,6.754,148.998
C02629=1141.105,110.542,-55.594,-179.162,6.753,148.999
C02630=1141.110,110.293,-55.574,-179.165,6.751,148.999
C02631=1141.115,110.044,-55.556,-179.168,6.749,149.000
C02632=1141.120,109.795,-55.537,-179.171,6.748,149.000
C02633=1141.124,109.545,-55.518,-179.173,6.747,149.001
C02634=1141.130,109.296,-55.499,-179.176,6.745,149.001
C02635=1141.134,109.046,-55.481,-179.178,6.744,149.001
C02636=1141.138,108.798,-55.462,-179.181,6.742,149.002
C02637=1141.144,108.548,-55.444,-179.184,6.740,149.002
C02638=1141.148,108.299,-55.424,-179.187,6.739,149.003
C02639=1141.154,108.049,-55.406,-179.189,6.737,149.003
C02640=1141.158,107.801,-55.387,-179.192,6.735,149.003
C02641=1141.163,107.551,-55.369,-179.195,6.734,149.004
C02642=1141.168,107.302,-55.350,-179.198,6.732,149.005
C02643=1141.173,107.053,-55.332,-179.201,6.731,149.005
C02644=1141.177,106.803,-55.313,-179.204,6.729,149.005
C02645=1141.183,106.554,-55.294,-179.206,6.727,149.006
C02646=1141.187,106.305,-55.276,-179.209,6.726,149.006
C02647=1141.191,106.056,-55.257,-179.212,6.724,149.007
C02648=1141.197,105.787,-55.237,-179.215,6.723,149.007
C02649=1141.202,105.519,-55.217,-179.218,6.721,149.008
C02650=1141.208,105.250,-55.197,-179.220,6.719,149.008
C02651=1141.213,104.983,-55.177,-179.223,6.718,149.008
C02652=1141.218,104.732,-55.158,-179.226,6.716,149.009
C02653=1141.223,104.483,-55.140,-179.229,6.715,149.009
C02654=1141.228,104.234,-55.122,-179.232,6.713,149.010
C02655=1141.232,103.985,-55.103,-179.235,6.711,149.010
C02656=1141.238,103.735,-55.085,-179.237,6.710,149.011
C02657=1141.242,103.486,-55.067,-179.240,6.708,149.011
C02658=1141.247,103.238,-55.048,-179.243,6.706,149.012
C02659=1141.251,102.988,-55.030,-179.246,6.705,149.012
C02660=1141.257,102.738,-55.011,-179.249,6.703,149.013
C02661=1141.262,102.489,-54.993,-179.251,6.701,149.013
C02662=1141.267,102.240,-54.975,-179.254,6.700,149.013
C02663=1141.271,101.991,-54.956,-179.256,6.699,149.014
C02664=1141.276,101.742,-54.938,-179.259,6.697,149.014
C02665=1141.281,101.492,-54.920,-179.262,6.696,149.015
C02666=1141.286,101.243,-54.902,-179.265,6.694,149.015
C02667=1141.291,100.994,-54.884,-179.268,6.693,149.016
C02668=1141.296,100.744,-54.865,-179.270,6.691,149.016
C02669=1141.300,100.495,-54.847,-179.273,6.689,149.017
C02670=1141.306,100.246,-54.828,-179.276,6.688,149.017
C02671=1141.311,99.997,-54.810,-179.279,6.686,149.017
C02672=1141.316,99.747,-54.792,-179.281,6.684,149.018
C02673=1141.320,99.498,-54.774,-179.284,6.684,149.018
C02674=1141.325,99.248,-54.756,-179.287,6.682,149.019
C02675=1141.330,98.999,-54.738,-179.289,6.680,149.019
C02676=1141.335,98.750,-54.720,-179.292,6.679,149.020
C02677=1141.340,98.501,-54.702,-179.295,6.677,149.020
C02678=1141.344,98.252,-54.684,-179.298,6.675,149.021
C02679=1141.350,98.001,-54.665,-179.301,6.674,149.021
C02680=1141.354,97.752,-54.647,-179.304,6.672,149.022
C02681=1141.359,97.503,-54.629,-179.306,6.671,149.022
C02682=1141.364,97.254,-54.611,-179.308,6.670,149.022
C02683=1141.369,97.005,-54.593,-179.311,6.668,149.023
C02684=1141.374,96.756,-54.575,-179.314,6.666,149.023
C02685=1141.379,96.506,-54.557,-179.317,6.665,149.024
C02686=1141.383,96.257,-54.539,-179.320,6.663,149.024
C02687=1141.388,96.007,-54.521,-179.323,6.662,149.025
C02688=1141.393,95.758,-54.503,-179.325,6.660,149.025
C02689=1141.398,95.509,-54.485,-179.328,6.659,149.026
C02690=1141.403,95.260,-54.467,-179.330,6.658,149.026
C02691=1141.408,95.011,-54.449,-179.333,6.656,149.027
C02692=1141.413,94.761,-54.431,-179.336,6.655,149.027
C02693=1141.418,94.512,-54.413,-179.339,6.653,149.027
C02694=1141.423,94.263,-54.396,-179.342,6.651,149.028
C02695=1141.428,94.013,-54.378,-179.344,6.650,149.028
C02696=1141.433,93.764,-54.360,-179.347,6.649,149.029
C02697=1141.437,93.514,-54.341,-179.350,6.647,149.029
C02698=1141.442,93.265,-54.323,-179.353,6.646,149.030
C02699=1141.447,93.016,-54.305,-179.355,6.644,149.030
C02700=1141.452,92.766,-54.288,-179.358,6.642,149.031
C02701=1141.457,92.517,-54.270,-179.361,6.641,149.031
C02702=1141.462,92.268,-54.252,-179.363,6.640,149.032
C02703=1141.467,92.019,-54.234,-179.366,6.639,149.032
C02704=1141.471,91.769,-54.217,-179.369,6.637,149.033
C02705=1141.476,91.520,-54.199,-179.372,6.635,149.033
C02706=1141.481,91.271,-54.181,-179.374,6.634,149.033
C02707=1141.486,91.022,-54.163,-179.378,6.632,149.034
C02708=1141.491,90.772,-54.146,-179.380,6.631,149.034
C02709=1141.496,90.523,-54.128,-179.382,6.630,149.035
C02710=1141.501,90.273,-54.110,-179.385,6.628,149.035
C02711=1141.506,90.024,-54.092,-179.388,6.626,149.036
C02712=1141.510,89.775,-54.076,-179.391,6.625,149.036
C02713=1141.515,89.526,-54.058,-179.393,6.624,149.037
C02714=1141.520,89.276,-54.040,-179.396,6.622,149.037
C02715=1141.526,89.027,-54.022,-179.399,6.621,149.038
C02716=1141.530,88.777,-54.004,-179.402,6.620,149.038
C02717=1141.536,88.528,-53.987,-179.405,6.618,149.039
C02718=1141.540,88.279,-53.970,-179.407,6.617,149.039
C02719=1141.545,88.030,-53.952,-179.410,6.615,149.040
C02720=1141.550,87.780,-53.935,-179.412,6.614,149.040
C02721=1141.555,87.531,-53.917,-179.416,6.612,149.041
C02722=1141.560,87.281,-53.899,-179.418,6.611,149.041
C02723=1141.564,87.032,-53.882,-179.420,6.610,149.041
C02724=1141.569,86.782,-53.865,-179.423,6.608,149.042
C02725=1141.574,86.533,-53.847,-179.426,6.606,149.042
C02726=1141.580,86.285,-53.829,-179.429,6.605,149.043
C02727=1141.584,86.035,-53.812,-179.432,6.604,149.043
C02728=1141.589,85.786,-53.794,-179.434,6.603,149.044
C02729=1141.594,85.536,-53.777,-179.437,6.601,149.044
C02730=1141.599,85.287,-53.760,-179.440,6.600,149.045
C02731=1141.604,85.037,-53.742,-179.443,6.598,149.045
C02732=1141.609,84.788,-53.724,-179.445,6.596,149.046
C02733=1141.614,84.538,-53.707,-179.448,6.595,149.046
C02734=1141.618,84.289,-53.691,-179.450,6.594,149.047
C02735=1141.623,84.040,-53.673,-179.454,6.593,149.047
C02736=1141.629,83.791,-53.656,-179.456,6.591,149.048
C02737=1141.633,83.542,-53.638,-179.458,6.590,149.048
C02738=1141.639,83.292,-53.621,-179.461,6.588,149.049
C02739=1141.644,83.042,-53.604,-179.464,6.587,149.049
C02740=1141.648,82.793,-53.586,-179.467,6.585,149.050
C02741=1141.653,82.544,-53.569,-179.469,6.584,149.050
C02742=1141.658,82.294,-53.551,-179.472,6.583,149.050
C02743=1141.663,82.045,-53.534,-179.475,6.582,149.051
C02744=1141.668,81.796,-53.518,-179.478,6.580,149.052
C02745=1141.673,81.547,-53.500,-179.480,6.579,149.052
C02746=1141.678,81.297,-53.483,-179.483,6.577,149.052
C02747=1141.683,81.047,-53.466,-179.486,6.576,149.053
C02748=1141.687,80.799,-53.448,-179.489,6.574,149.053
C02749=1141.692,80.549,-53.431,-179.491,6.574,149.054
C02750=1141.698,80.300,-53.415,-179.494,6.572,149.054
C02751=1141.703,80.050,-53.397,-179.496,6.570,149.055
C02752=1141.708,79.782,-53.378,-179.500,6.569,149.055
C02753=1141.713,79.514,-53.360,-179.502,6.567,149.056
C02754=1141.718,79.245,-53.342,-179.506,6.566,149.056
C02755=1141.723,78.977,-53.323,-179.508,6.564,149.057
C02756=1141.729,78.728,-53.307,-179.511,6.563,149.057
C02757=1141.733,78.478,-53.290,-179.514,6.562,149.058
C02758=1141.739,78.228,-53.273,-179.517,6.560,149.058
C02759=1141.744,77.979,-53.255,-179.519,6.559,149.059
C02760=1141.748,77.730,-53.238,-179.521,6.558,149.059
C02761=1141.754,77.480,-53.221,-179.525,6.557,149.060
C02762=1141.758,77.231,-53.204,-179.527,6.555,149.060
C02763=1141.763,76.982,-53.188,-179.530,6.553,149.061
C02764=1141.768,76.732,-53.171,-179.532,6.552,149.061
C02765=1141.773,76.483,-53.154,-179.536,6.551,149.062
C02766=1141.778,76.234,-53.136,-179.538,6.550,149.062
C02767=1141.782,75.984,-53.120,-179.540,6.549,149.063
C02768=1141.788,75.735,-53.103,-179.543,6.547,149.063
C02769=1141.793,75.486,-53.086,-179.546,6.546,149.064
C02770=1141.798,75.236,-53.069,-179.549,6.544,149.064
C02771=1141.802,74.986,-53.052,-179.551,6.543,149.065
C02772=1141.808,74.738,-53.036,-179.554,6.542,149.065
C02773=1141.813,74.488,-53.018,-179.557,6.540,149.066
C02774=1141.817,74.238,-53.002,-179.559,6.539,149.066
C02775=1141.823,73.989,-52.985,-179.562,6.538,149.067
C02776=1141.828,73.740,-52.968,-179.565,6.536,149.067
C02777=1141.832,73.490,-52.952,-179.568,6.536,149.068
C02778=1141.837,73.241,-52.934,-179.570,6.534,149.068
C02779=1141.842,72.992,-52.918,-179.573,6.532,149.069
C02780=1141.848,72.742,-52.901,-179.576,6.532,149.069
C02781=1141.852,72.492,-52.884,-179.578,6.530,149.070
C02782=1141.857,72.244,-52.868,-179.581,6.528,149.070
C02783=1141.862,71.994,-52.851,-179.584,6.527,149.071
C02784=1141.867,71.744,-52.834,-179.587,6.526,149.071
C02785=1141.872,71.496,-52.818,-179.589,6.525,149.072
C02786=1141.877,71.246,-52.800,-179.592,6.523,149.072
C02787=1141.882,70.996,-52.784,-179.595,6.523,149.073
C02788=1141.887,70.747,-52.768,-179.597,6.521,149.073
C02789=1141.892,70.497,-52.751,-179.600,6.519,149.074
C02790=1141.897,70.248,-52.734,-179.602,6.518,149.074
C02791=1141.902,69.999,-52.718,-179.606,6.517,149.075
C02792=1141.906,69.749,-52.701,-179.608,6.515,149.075
C02793=1141.912,69.500,-52.684,-179.610,6.515,149.076
C02794=1141.917,69.251,-52.668,-179.614,6.513,149.076
C02795=1141.921,69.001,-52.652,-179.616,6.512,149.077
C02796=1141.926,68.752,-52.635,-179.619,6.511,149.077
C02797=1141.932,68.502,-52.618,-179.621,6.509,149.077
C02798=1141.937,68.253,-52.602,-179.625,6.508,149.078
C02799=1141.941,68.004,-52.585,-179.627,6.507,149.079
C02800=1141.946,67.754,-52.569,-179.629,6.505,149.079
C02801=1141.952,67.505,-52.552,-179.633,6.504,149.080
C02802=1141.956,67.255,-52.536,-179.635,6.503,149.080
C02803=1141.961,67.006,-52.519,-179.638,6.502,149.081
C02804=1141.966,66.756,-52.503,-179.640,6.501,149.081
C02805=1141.971,66.507,-52.487,-179.643,6.499,149.082
C02806=1141.976,66.258,-52.470,-179.646,6.498,149.082
C02807=1141.981,66.008,-52.454,-179.648,6.497,149.082
C02808=1141.986,65.759,-52.437,-179.651,6.496,149.083
C02809=1141.991,65.509,-52.421,-179.654,6.494,149.084
C02810=1141.996,65.260,-52.405,-179.656,6.493,149.084
C02811=1142.001,65.010,-52.389,-179.659,6.492,149.085
C02812=1142.006,64.762,-52.372,-179.662,6.490,149.085
C02813=1142.011,64.511,-52.356,-179.664,6.489,149.086
C02814=1142.016,64.262,-52.339,-179.667,6.488,149.086
C02815=1142.021,64.013,-52.323,-179.669,6.487,149.087
C02816=1142.026,63.764,-52.307,-179.672,6.486,149.087
C02817=1142.031,63.514,-52.290,-179.675,6.484,149.088
C02818=1142.036,63.265,-52.275,-179.678,6.483,149.088
C02819=1142.041,63.015,-52.258,-179.680,6.482,149.089
C02820=1142.046,62.766,-52.242,-179.683,6.480,149.089
C02821=1142.050,62.516,-52.226,-179.686,6.480,149.090
C02822=1142.055,62.268,-52.210,-179.689,6.478,149.090
C02823=1142.060,62.017,-52.194,-179.691,6.477,149.091
C02824=1142.065,61.769,-52.177,-179.694,6.476,149.091
C02825=1142.071,61.518,-52.161,-179.697,6.474,149.092
C02826=1142.076,61.269,-52.145,-179.699,6.473,149.092
C02827=1142.081,61.019,-52.129,-179.702,6.472,149.093
C02828=1142.086,60.771,-52.112,-179.704,6.471,149.093
C02829=1142.091,60.520,-52.096,-179.707,6.470,149.094
C02830=1142.096,60.272,-52.080,-179.710,6.468,149.094
C02831=1142.101,60.022,-52.064,-179.712,6.467,149.095
C02832=1142.106,59.773,-52.048,-179.715,6.466,149.095
C02833=1142.111,59.523,-52.032,-179.717,6.465,149.096
C02834=1142.115,59.274,-52.015,-179.720,6.464,149.096
C02835=1142.121,59.025,-52.000,-179.723,6.462,149.097
C02836=1142.126,58.774,-51.984,-179.725,6.461,149.097
C02837=1142.131,58.526,-51.968,-179.729,6.460,149.098
C02838=1142.136,58.276,-51.952,-179.731,6.459,149.098
C02839=1142.140,58.027,-51.936,-179.734,6.457,149.099
C02840=1142.145,57.778,-51.920,-179.736,6.457,149.099
C02841=1142.150,57.528,-51.904,-179.739,6.455,149.100
C02842=1142.155,57.279,-51.888,-179.742,6.454,149.100
C02843=1142.160,57.029,-51.873,-179.744,6.453,149.101
C02844=1142.165,56.779,-51.857,-179.747,6.452,149.101
C02845=1142.170,56.530,-51.840,-179.749,6.451,149.102
C02846=1142.175,56.280,-51.824,-179.752,6.449,149.103
C02847=1142.181,56.031,-51.809,-179.755,6.449,149.103
C02848=1142.186,55.782,-51.793,-179.757,6.447,149.103
C02849=1142.190,55.532,-51.776,-179.761,6.446,149.104
C02850=1142.196,55.283,-51.761,-179.763,6.445,149.104
C02851=1142.200,55.034,-51.746,-179.765,6.443,149.105
C02852=1142.205,54.784,-51.729,-179.768,6.443,149.106
C02853=1142.210,54.535,-51.714,-179.771,6.441,149.106
C02854=1142.216,54.285,-51.698,-179.773,6.440,149.106
C02855=1142.220,54.035,-51.682,-179.776,6.439,149.107
C02856=1142.226,53.767,-51.665,-179.779,6.437,149.108
C02857=1142.232,53.498,-51.648,-179.782,6.437,149.108
C02858=1142.237,53.230,-51.631,-179.784,6.435,149.109
C02859=1142.242,52.962,-51.615,-179.788,6.434,149.109
C02860=1142.247,52.711,-51.599,-179.790,6.433,149.110
C02861=1142.252,52.462,-51.583,-179.793,6.431,149.110
C02862=1142.257,52.213,-51.568,-179.796,6.430,149.111
C02863=1142.262,51.963,-51.552,-179.798,6.429,149.111
C02864=1142.267,51.714,-51.536,-179.801,6.428,149.112
C02865=1142.272,51.465,-51.520,-179.803,6.427,149.112
C02866=1142.277,51.215,-51.505,-179.806,6.426,149.113
C02867=1142.282,50.965,-51.489,-179.808,6.425,149.113
C02868=1142.287,50.716,-51.474,-179.812,6.423,149.114
C02869=1142.292,50.467,-51.458,-179.814,6.423,149.114
C02870=1142.297,50.217,-51.442,-179.816,6.421,149.115
C02871=1142.302,49.967,-51.427,-179.819,6.421,149.116
C02872=1142.307,49.718,-51.412,-179.822,6.419,149.116
C02873=1142.312,49.469,-51.396,-179.824,6.418,149.116
C02874=1142.317,49.219,-51.380,-179.827,6.417,149.117
C02875=1142.323,48.969,-51.364,-179.829,6.416,149.118
C02876=1142.327,48.720,-51.349,-179.833,6.415,149.118
C02877=1142.333,48.471,-51.334,-179.835,6.414,149.119
C02878=1142.337,48.221,-51.318,-179.838,6.412,149.119
C02879=1142.342,47.971,-51.303,-179.840,6.412,149.120
C02880=1142.347,47.722,-51.287,-179.843,6.410,149.120
C02881=1142.353,47.473,-51.272,-179.845,6.409,149.121
C02882=1142.357,47.224,-51.257,-179.848,6.408,149.121
C02883=1142.362,46.973,-51.241,-179.850,6.407,149.122
C02884=1142.368,46.724,-51.225,-179.853,6.405,149.122
C02885=1142.372,46.475,-51.210,-179.856,6.405,149.123
C02886=1142.378,46.226,-51.195,-179.859,6.403,149.123
C02887=1142.382,45.976,-51.179,-179.861,6.403,149.124
C02888=1142.387,45.726,-51.164,-179.864,6.401,149.124
C02889=1142.393,45.477,-51.148,-179.866,6.400,149.125
C02890=1142.397,45.228,-51.133,-179.869,6.399,149.125
C02891=1142.403,44.979,-51.118,-179.872,6.398,149.126
C02892=1142.408,44.729,-51.103,-179.874,6.397,149.127
C02893=1142.412,44.479,-51.087,-179.877,6.396,149.127
C02894=1142.418,44.229,-51.072,-179.880,6.395,149.128
C02895=1142.422,43.980,-51.057,-179.882,6.394,149.128
C02896=1142.428,43.731,-51.041,-179.885,6.393,149.129
C02897=1142.432,43.482,-51.026,-179.887,6.392,149.129
C02898=1142.438,43.232,-51.011,-179.890,6.390,149.130
C02899=1142.443,42.983,-50.996,-179.893,6.390,149.130
C02900=1142.448,42.732,-50.980,-179.895,6.388,149.131
C02901=1142.453,42.483,-50.965,-179.898,6.387,149.131
C02902=1142.458,42.234,-50.950,-179.901,6.386,149.132
C02903=1142.463,41.984,-50.935,-179.903,6.385,149.132
C02904=1142.468,41.735,-50.920,-179.906,6.383,149.133
C02905=1142.473,41.485,-50.904,-179.908,6.383,149.133
C02906=1142.478,41.236,-50.890,-179.911,6.381,149.134
C02907=1142.484,40.986,-50.874,-179.914,6.381,149.135
C02908=1142.488,40.737,-50.859,-179.916,6.380,149.135
C02909=1142.493,40.487,-50.843,-179.919,6.378,149.135
C02910=1142.498,40.237,-50.829,-179.921,6.378,149.136
C02911=1142.503,39.988,-50.814,-179.924,6.376,149.137
C02912=1142.508,39.739,-50.799,-179.926,6.375,149.137
C02913=1142.513,39.489,-50.784,-179.930,6.374,149.138
C02914=1142.518,39.240,-50.769,-179.932,6.373,149.138
C02915=1142.523,38.991,-50.754,-179.935,6.372,149.139
C02916=1142.529,38.741,-50.739,-179.937,6.371,149.139
C02917=1142.533,38.492,-50.724,-179.940,6.370,149.140
C02918=1142.539,38.242,-50.709,-179.943,6.369,149.140
C02919=1142.544,37.993,-50.694,-179.945,6.368,149.141
C02920=1142.548,37.743,-50.679,-179.947,6.367,149.141
C02921=1142.554,37.493,-50.664,-179.950,6.366,149.142
C02922=1142.559,37.244,-50.649,-179.953,6.365,149.142
C02923=1142.564,36.994,-50.634,-179.956,6.364,149.143
C02924=1142.569,36.745,-50.619,-179.958,6.362,149.144
C02925=1142.574,36.496,-50.604,-179.960,6.362,149.144
C02926=1142.579,36.246,-50.589,-179.963,6.361,149.145
C02927=1142.584,35.997,-50.574,-179.966,6.360,149.145
C02928=1142.590,35.747,-50.560,-179.968,6.359,149.146
C02929=1142.594,35.498,-50.545,-179.971,6.357,149.146
C02930=1142.599,35.248,-50.530,-179.973,6.357,149.147
C02931=1142.605,34.999,-50.515,-179.977,6.355,149.147
C02932=1142.610,34.749,-50.500,-179.979,6.355,149.148
C02933=1142.614,34.500,-50.485,-179.981,6.354,149.148
C02934=1142.620,34.250,-50.471,-179.984,6.352,149.149
C02935=1142.625,34.000,-50.456,-179.986,6.352,149.149
C02936=1142.630,33.751,-50.441,-179.989,6.350,149.150
C02937=1142.635,33.501,-50.426,-179.992,6.350,149.151
C02938=1142.640,33.252,-50.411,-179.994,6.349,149.151
C02939=1142.645,33.002,-50.397,-179.997,6.347,149.152
C02940=1142.650,32.753,-50.382,-179.999,6.347,149.152
C02941=1142.655,32.503,-50.367,179.998,6.345,149.153
C02942=1142.660,32.254,-50.353,179.995,6.345,149.153
C02943=1142.665,32.004,-50.338,179.993,6.344,149.154
C02944=1142.670,31.755,-50.324,179.990,6.342,149.154
C02945=1142.675,31.505,-50.308,179.988,6.342,149.155
C02946=1142.680,31.256,-50.294,179.985,6.340,149.155
C02947=1142.685,31.006,-50.280,179.982,6.340,149.156
C02948=1142.690,30.757,-50.265,179.980,6.339,149.156
C02949=1142.695,30.507,-50.250,179.977,6.337,149.157
C02950=1142.700,30.257,-50.235,179.975,6.337,149.158
C02951=1142.705,30.008,-50.220,179.972,6.335,149.158
C02952=1142.711,29.759,-50.207,179.969,6.335,149.159
C02953=1142.716,29.509,-50.192,179.967,6.334,149.159
C02954=1142.721,29.259,-50.177,179.964,6.332,149.160
C02955=1142.726,29.010,-50.162,179.962,6.332,149.160
C02956=1142.731,28.760,-50.148,179.959,6.331,149.161
C02957=1142.736,28.511,-50.134,179.957,6.329,149.161
C02958=1142.741,28.261,-50.120,179.954,6.329,149.162
C02959=1142.745,28.012,-50.105,179.951,6.327,149.162
C02960=1142.752,27.742,-50.089,179.949,6.327,149.163
C02961=1142.757,27.474,-50.074,179.946,6.325,149.163
C02962=1142.762,27.205,-50.058,179.943,6.325,149.164
C02963=1142.768,26.936,-50.043,179.940,6.323,149.165
C02964=1142.773,26.687,-50.028,179.938,6.323,149.165
C02965=1142.778,26.437,-50.013,179.935,6.321,149.166
C02966=1142.783,26.187,-49.999,179.932,6.320,149.166
C02967=1142.788,25.937,-49.985,179.930,6.320,149.167
C02968=1142.794,25.688,-49.971,179.927,6.318,149.167
C02969=1142.799,25.439,-49.956,179.925,6.318,149.168
C02970=1142.803,25.190,-49.941,179.923,6.317,149.168
C02971=1142.808,24.940,-49.927,179.919,6.316,149.169
C02972=1142.813,24.690,-49.913,179.917,6.315,149.170
C02973=1142.818,24.440,-49.899,179.915,6.314,149.170
C02974=1142.824,24.191,-49.885,179.912,6.313,149.171
C02975=1142.829,23.942,-49.870,179.910,6.312,149.171
C02976=1142.834,23.692,-49.856,179.907,6.311,149.172
C02977=1142.839,23.442,-49.842,179.904,6.310,149.172
C02978=1142.844,23.192,-49.827,179.902,6.309,149.173
C02979=1142.850,22.943,-49.813,179.899,6.308,149.173
C02980=1142.855,22.694,-49.799,179.897,6.307,149.174
C02981=1142.860,22.444,-49.784,179.894,6.306,149.175
C02982=1142.865,22.194,-49.770,179.892,6.306,149.175
C02983=1142.870,21.945,-49.756,179.889,6.304,149.175
C02984=1142.875,21.695,-49.742,179.886,6.303,149.176
C02985=1142.880,21.446,-49.728,179.884,6.303,149.177
C02986=1142.885,21.196,-49.713,179.881,6.301,149.177
C02987=1142.889,20.947,-49.700,179.879,6.301,149.178
C02988=1142.895,20.698,-49.686,179.877,6.300,149.178
C02989=1142.900,20.448,-49.672,179.873,6.299,149.179
C02990=1142.905,20.198,-49.657,179.871,6.298,149.179
C02991=1142.910,19.948,-49.643,179.869,6.297,149.180
C02992=1142.915,19.699,-49.629,179.866,6.296,149.180
C02993=1142.920,19.450,-49.615,179.864,6.295,149.181
C02994=1142.925,19.200,-49.601,179.861,6.294,149.182
C02995=1142.931,18.951,-49.587,179.858,6.293,149.182
C02996=1142.936,18.701,-49.572,179.856,6.292,149.183
C02997=1142.941,18.452,-49.558,179.853,6.291,149.183
C02998=1142.946,18.201,-49.545,179.851,6.291,149.184
C02999=1142.951,17.952,-49.531,179.848,6.289,149.184
C03000=1142.956,17.703,-49.516,179.846,6.289,149.185
C03001=1142.961,17.453,-49.503,179.843,6.288,149.185
C03002=1142.966,17.204,-49.489,179.840,6.287,149.186
C03003=1142.971,16.954,-49.474,179.838,6.286,149.186
C03004=1142.976,16.705,-49.460,179.836,6.285,149.187
C03005=1142.982,16.455,-49.447,179.833,6.284,149.188
C03006=1142.987,16.205,-49.433,179.830,6.283,149.188
C03007=1142.992,15.956,-49.418,179.828,6.282,149.189
C03008=1142.997,15.707,-49.405,179.826,6.282,149.189
C03009=1143.002,15.457,-49.391,179.823,6.280,149.190
C03010=1143.007,15.207,-49.377,179.820,6.280,149.190
C03011=1143.012,14.958,-49.363,179.818,6.279,149.191
C03012=1143.017,14.708,-49.349,179.815,6.277,149.191
C03013=1143.022,14.458,-49.335,179.812,6.277,149.192
C03014=1143.028,14.209,-49.322,179.810,6.276,149.193
C03015=1143.032,13.959,-49.308,179.808,6.275,149.193
C03016=1143.037,13.710,-49.294,179.805,6.274,149.194
C03017=1143.043,13.460,-49.280,179.803,6.273,149.194
C03018=1143.048,13.210,-49.266,179.800,6.273,149.195
C03019=1143.052,12.961,-49.253,179.798,6.272,149.195
C03020=1143.058,12.712,-49.239,179.795,6.270,149.196
C03021=1143.063,12.462,-49.225,179.792,6.270,149.196
C03022=1143.069,12.213,-49.211,179.790,6.269,149.197
C03023=1143.073,11.963,-49.197,179.787,6.268,149.198
C03024=1143.078,11.713,-49.184,179.785,6.267,149.198
C03025=1143.084,11.464,-49.170,179.783,6.266,149.199
C03026=1143.089,11.214,-49.156,179.780,6.266,149.199
C03027=1143.094,10.965,-49.143,179.777,6.264,149.200
C03028=1143.099,10.715,-49.129,179.775,6.264,149.200
C03029=1143.104,10.465,-49.115,179.772,6.263,149.201
C03030=1143.109,10.216,-49.102,179.770,6.262,149.201
C03031=1143.114,9.966,-49.088,179.767,6.261,149.202
C03032=1143.120,9.717,-49.074,179.765,6.260,149.202
C03033=1143.125,9.467,-49.060,179.762,6.260,149.203
C03034=1143.130,9.218,-49.048,179.760,6.259,149.204
C03035=1143.135,8.968,-49.033,179.757,6.257,149.204
C03036=1143.141,8.718,-49.020,179.754,6.257,149.205
C03037=1143.145,8.469,-49.006,179.752,6.256,149.205
C03038=1143.150,8.219,-48.993,179.750,6.256,149.206
C03039=1143.156,7.970,-48.979,179.747,6.254,149.206
C03040=1143.160,7.720,-48.966,179.745,6.253,149.207
C03041=1143.166,7.471,-48.952,179.742,6.253,149.207
C03042=1143.170,7.221,-48.939,179.740,6.252,149.208
C03043=1143.176,6.972,-48.925,179.737,6.252,149.209
C03044=1143.181,6.721,-48.912,179.734,6.250,149.209
C03045=1143.186,6.473,-48.898,179.732,6.249,149.210
C03046=1143.191,6.222,-48.885,179.730,6.249,149.210
C03047=1143.196,5.974,-48.871,179.727,6.248,149.211
C03048=1143.201,5.723,-48.858,179.724,6.247,149.211
C03049=1143.207,5.474,-48.845,179.722,6.246,149.212
C03050=1143.211,5.224,-48.831,179.719,6.245,149.213
C03051=1143.217,4.975,-48.818,179.717,6.245,149.213
C03052=1143.221,4.725,-48.804,179.715,6.244,149.213
C03053=1143.227,4.476,-48.791,179.712,6.243,149.214
C03054=1143.232,4.226,-48.778,179.710,6.242,149.215
C03055=1143.237,3.977,-48.764,179.707,6.241,149.215
C03056=1143.243,3.726,-48.751,179.705,6.240,149.216
C03057=1143.247,3.478,-48.737,179.702,6.239,149.216
C03058=1143.253,3.227,-48.724,179.699,6.238,149.217
C03059=1143.258,2.978,-48.711,179.697,6.238,149.217
C03060=1143.263,2.729,-48.697,179.695,6.237,149.218
C03061=1143.268,2.479,-48.684,179.692,6.236,149.219
C03062=1143.274,2.229,-48.671,179.689,6.235,149.219
C03063=1143.278,1.979,-48.658,179.687,6.234,149.220
C03064=1143.284,1.710,-48.643,179.684,6.234,149.220
C03065=1143.290,1.440,-48.629,179.682,6.233,149.221
C03066=1143.295,1.171,-48.615,179.679,6.232,149.222
C03067=1143.301,0.901,-48.600,179.677,6.231,149.222
C03068=1143.305,0.653,-48.587,179.674,6.231,149.223
C03069=1143.311,0.403,-48.574,179.671,6.229,149.223
C03070=1143.316,0.153,-48.561,179.669,6.229,149.224
C03071=1143.322,-0.097,-48.548,179.666,6.228,149.224
C03072=1143.326,-0.347,-48.535,179.664,6.227,149.225
C03073=1143.332,-0.596,-48.521,179.662,6.227,149.225
C03074=1143.337,-0.845,-48.508,179.659,6.225,149.226
C03075=1143.342,-1.095,-48.495,179.656,6.225,149.227
C03076=1143.347,-1.345,-48.482,179.654,6.224,149.227
C03077=1143.352,-1.595,-48.469,179.652,6.223,149.228
C03078=1143.357,-1.844,-48.455,179.649,6.222,149.228
C03079=1143.362,-2.093,-48.443,179.647,6.222,149.229
C03080=1143.368,-2.343,-48.429,179.644,6.220,149.229
C03081=1143.373,-2.593,-48.416,179.642,6.220,149.230
C03082=1143.378,-2.842,-48.404,179.639,6.219,149.231
C03083=1143.383,-3.092,-48.390,179.637,6.218,149.231
C03084=1143.388,-3.342,-48.378,179.634,6.218,149.231
C03085=1143.392,-3.591,-48.364,179.632,6.217,149.232
C03086=1143.398,-3.841,-48.351,179.629,6.216,149.233
C03087=1143.403,-4.090,-48.338,179.626,6.215,149.233
C03088=1143.409,-4.340,-48.325,179.624,6.214,149.234
C03089=1143.414,-4.590,-48.312,179.622,6.214,149.234
C03090=1143.419,-4.839,-48.299,179.619,6.213,149.235
C03091=1143.424,-5.089,-48.286,179.617,6.212,149.235
C03092=1143.429,-5.339,-48.273,179.615,6.212,149.236
C03093=1143.435,-5.588,-48.261,179.612,6.210,149.237
C03094=1143.440,-5.838,-48.247,179.610,6.209,149.237
C03095=1143.445,-6.088,-48.235,179.607,6.209,149.238
C03096=1143.450,-6.337,-48.222,179.605,6.208,149.238
C03097=1143.455,-6.586,-48.209,179.602,6.208,149.239
C03098=1143.460,-6.837,-48.196,179.600,6.207,149.239
C03099=1143.466,-7.086,-48.183,179.597,6.206,149.240
C03100=1143.471,-7.335,-48.171,179.594,6.205,149.241
C03101=1143.476,-7.585,-48.157,179.592,6.204,149.241
C03102=1143.481,-7.835,-48.144,179.590,6.204,149.242
C03103=1143.486,-8.084,-48.132,179.587,6.203,149.242
C03104=1143.491,-8.333,-48.119,179.585,6.203,149.243
C03105=1143.497,-8.584,-48.106,179.583,6.202,149.243
C03106=1143.502,-8.833,-48.093,179.580,6.201,149.244
C03107=1143.507,-9.082,-48.080,179.577,6.200,149.244
C03108=1143.512,-9.332,-48.068,179.575,6.199,149.245
C03109=1143.516,-9.582,-48.055,179.572,6.198,149.246
C03110=1143.522,-9.831,-48.042,179.570,6.198,149.246
C03111=1143.527,-10.081,-48.029,179.568,6.197,149.247
C03112=1143.533,-10.331,-48.017,179.565,6.196,149.247
C03113=1143.537,-10.581,-48.004,179.563,6.196,149.248
C03114=1143.542,-10.830,-47.992,179.561,6.195,149.248
C03115=1143.548,-11.080,-47.978,179.558,6.194,149.249
C03116=1143.553,-11.329,-47.966,179.555,6.193,149.250
C03117=1143.558,-11.579,-47.953,179.553,6.192,149.250
C03118=1143.563,-11.828,-47.940,179.551,6.192,149.250
C03119=1143.569,-12.078,-47.928,179.548,6.191,149.251
C03120=1143.574,-12.327,-47.916,179.546,6.190,149.252
C03121=1143.579,-12.578,-47.902,179.543,6.190,149.252
C03122=1143.584,-12.827,-47.890,179.541,6.189,149.253
C03123=1143.589,-13.076,-47.877,179.539,6.188,149.253
C03124=1143.595,-13.326,-47.865,179.536,6.187,149.254
C03125=1143.600,-13.576,-47.853,179.533,6.186,149.254
C03126=1143.605,-13.825,-47.840,179.531,6.186,149.255
C03127=1143.609,-14.075,-47.827,179.529,6.185,149.256
C03128=1143.615,-14.325,-47.815,179.526,6.184,149.256
C03129=1143.621,-14.575,-47.802,179.524,6.184,149.257
C03130=1143.626,-14.824,-47.789,179.522,6.183,149.257
C03131=1143.631,-15.073,-47.777,179.519,6.183,149.258
C03132=1143.636,-15.324,-47.764,179.517,6.182,149.258
C03133=1143.641,-15.573,-47.752,179.515,6.181,149.259
C03134=1143.646,-15.823,-47.739,179.512,6.181,149.260
C03135=1143.651,-16.072,-47.727,179.509,6.179,149.260
C03136=1143.657,-16.322,-47.715,179.506,6.179,149.261
C03137=1143.662,-16.571,-47.702,179.504,6.178,149.261
C03138=1143.667,-16.820,-47.690,179.502,6.177,149.262
C03139=1143.672,-17.071,-47.677,179.499,6.177,149.262
C03140=1143.677,-17.320,-47.665,179.497,6.176,149.263
C03141=1143.682,-17.570,-47.653,179.495,6.175,149.264
C03142=1143.687,-17.820,-47.640,179.492,6.175,149.264
C03143=1143.692,-18.069,-47.628,179.490,6.174,149.265
C03144=1143.698,-18.319,-47.616,179.488,6.173,149.265
C03145=1143.703,-18.568,-47.603,179.485,6.173,149.266
C03146=1143.708,-18.817,-47.591,179.483,6.172,149.266
C03147=1143.714,-19.067,-47.579,179.481,6.171,149.267
C03148=1143.718,-19.317,-47.566,179.478,6.171,149.267
C03149=1143.723,-19.567,-47.554,179.475,6.169,149.268
C03150=1143.729,-19.817,-47.541,179.473,6.169,149.268
C03151=1143.734,-20.067,-47.529,179.470,6.168,149.269
C03152=1143.739,-20.316,-47.517,179.468,6.167,149.270
C03153=1143.744,-20.565,-47.504,179.465,6.167,149.270
C03154=1143.750,-20.815,-47.492,179.463,6.166,149.271
C03155=1143.755,-21.065,-47.480,179.461,6.165,149.271
C03156=1143.760,-21.314,-47.468,179.458,6.165,149.272
C03157=1143.765,-21.564,-47.455,179.456,6.164,149.272
C03158=1143.771,-21.814,-47.443,179.454,6.164,149.273
C03159=1143.776,-22.063,-47.431,179.451,6.163,149.274
C03160=1143.781,-22.313,-47.419,179.449,6.162,149.274
C03161=1143.786,-22.562,-47.406,179.447,6.162,149.275
C03162=1143.792,-22.812,-47.394,179.444,6.161,149.275
C03163=1143.796,-23.062,-47.381,179.442,6.161,149.276
C03164=1143.802,-23.312,-47.369,179.440,6.160,149.276
C03165=1143.807,-23.562,-47.358,179.437,6.159,149.277
C03166=1143.812,-23.811,-47.346,179.435,6.159,149.278
C03167=1143.817,-24.061,-47.334,179.432,6.158,149.278
C03168=1143.824,-24.331,-47.320,179.429,6.157,149.279
C03169=1143.829,-24.601,-47.307,179.427,6.156,149.279
C03170=1143.834,-24.871,-47.294,179.424,6.155,149.280
C03171=1143.840,-25.141,-47.281,179.422,6.155,149.281
C03172=1143.845,-25.391,-47.269,179.420,6.154,149.281
C03173=1143.851,-25.640,-47.257,179.417,6.153,149.282
C03174=1143.856,-25.890,-47.245,179.415,6.153,149.282
C03175=1143.861,-26.139,-47.232,179.412,6.152,149.283
C03176=1143.866,-26.389,-47.221,179.410,6.152,149.283
C03177=1143.871,-26.639,-47.209,179.408,6.151,149.284
C03178=1143.876,-26.888,-47.196,179.405,6.150,149.284
C03179=1143.882,-27.138,-47.185,179.403,6.150,149.285
C03180=1143.887,-27.388,-47.173,179.401,6.149,149.286
C03181=1143.892,-27.637,-47.161,179.398,6.148,149.286
C03182=1143.897,-27.887,-47.149,179.396,6.148,149.287
C03183=1143.902,-28.137,-47.137,179.394,6.147,149.287
C03184=1143.908,-28.386,-47.124,179.391,6.147,149.288
C03185=1143.913,-28.636,-47.112,179.389,6.146,149.288
C03186=1143.918,-28.886,-47.101,179.386,6.145,149.289
C03187=1143.923,-29.136,-47.089,179.384,6.145,149.289
C03188=1143.928,-29.385,-47.077,179.382,6.144,149.290
C03189=1143.934,-29.635,-47.065,179.379,6.143,149.291
C03190=1143.938,-29.885,-47.053,179.377,6.143,149.291
C03191=1143.944,-30.135,-47.042,179.374,6.142,149.292
C03192=1143.949,-30.384,-47.029,179.372,6.141,149.292
C03193=1143.955,-30.633,-47.017,179.370,6.141,149.293
C03194=1143.960,-30.883,-47.006,179.367,6.140,149.293
C03195=1143.965,-31.133,-46.994,179.365,6.139,149.294
C03196=1143.971,-31.383,-46.982,179.363,6.139,149.294
C03197=1143.975,-31.632,-46.970,179.360,6.138,149.295
C03198=1143.980,-31.882,-46.958,179.358,6.137,149.296
C03199=1143.986,-32.131,-46.947,179.355,6.137,149.296
C03200=1143.990,-32.381,-46.935,179.353,6.136,149.297
C03201=1143.996,-32.631,-46.923,179.351,6.135,149.297
C03202=1144.001,-32.881,-46.912,179.348,6.135,149.298
C03203=1144.007,-33.130,-46.899,179.346,6.134,149.298
C03204=1144.012,-33.379,-46.888,179.343,6.134,149.299
C03205=1144.017,-33.629,-46.876,179.341,6.133,149.300
C03206=1144.023,-33.879,-46.864,179.339,6.132,149.300
C03207=1144.027,-34.129,-46.853,179.336,6.132,149.301
C03208=1144.033,-34.379,-46.841,179.334,6.131,149.301
C03209=1144.037,-34.628,-46.830,179.332,6.131,149.302
C03210=1144.043,-34.878,-46.818,179.329,6.130,149.302
C03211=1144.049,-35.127,-46.806,179.327,6.129,149.303
C03212=1144.054,-35.377,-46.795,179.324,6.129,149.304
C03213=1144.059,-35.626,-46.782,179.322,6.128,149.304
C03214=1144.064,-35.876,-46.771,179.320,6.127,149.305
C03215=1144.069,-36.126,-46.759,179.317,6.127,149.305
C03216=1144.074,-36.376,-46.747,179.315,6.126,149.306
C03217=1144.080,-36.625,-46.737,179.313,6.125,149.306
C03218=1144.085,-36.875,-46.725,179.310,6.125,149.307
C03219=1144.090,-37.125,-46.713,179.308,6.124,149.307
C03220=1144.095,-37.374,-46.701,179.306,6.123,149.308
C03221=1144.100,-37.624,-46.690,179.303,6.123,149.309
C03222=1144.105,-37.874,-46.678,179.301,6.122,149.309
C03223=1144.111,-38.123,-46.667,179.299,6.121,149.310
C03224=1144.117,-38.373,-46.655,179.296,6.121,149.310
C03225=1144.121,-38.623,-46.644,179.294,6.120,149.311
C03226=1144.127,-38.873,-46.632,179.292,6.120,149.311
C03227=1144.131,-39.122,-46.620,179.290,6.120,149.312
C03228=1144.137,-39.371,-46.609,179.287,6.119,149.313
C03229=1144.142,-39.622,-46.598,179.285,6.118,149.313
C03230=1144.148,-39.872,-46.586,179.282,6.118,149.314
C03231=1144.153,-40.121,-46.575,179.280,6.117,149.314
C03232=1144.159,-40.370,-46.564,179.278,6.116,149.315
C03233=1144.163,-40.620,-46.552,179.275,6.116,149.315
C03234=1144.169,-40.870,-46.540,179.273,6.115,149.316
C03235=1144.173,-41.120,-46.529,179.271,6.114,149.316
C03236=1144.179,-41.369,-46.518,179.268,6.114,149.317
C03237=1144.184,-41.619,-46.506,179.266,6.113,149.318
C03238=1144.190,-41.868,-46.494,179.263,6.113,149.318
C03239=1144.195,-42.119,-46.484,179.261,6.112,149.319
C03240=1144.201,-42.368,-46.472,179.259,6.111,149.319
C03241=1144.205,-42.618,-46.461,179.256,6.111,149.320
C03242=1144.211,-42.868,-46.449,179.255,6.111,149.320
C03243=1144.215,-43.117,-46.438,179.253,6.110,149.321
C03244=1144.221,-43.366,-46.426,179.250,6.110,149.322
C03245=1144.226,-43.617,-46.416,179.248,6.109,149.322
C03246=1144.231,-43.866,-46.405,179.245,6.108,149.323
C03247=1144.237,-44.116,-46.393,179.243,6.108,149.323
C03248=1144.242,-44.365,-46.382,179.241,6.107,149.324
C03249=1144.247,-44.615,-46.370,179.238,6.107,149.324
C03250=1144.252,-44.865,-46.359,179.236,6.106,149.325
C03251=1144.258,-45.115,-46.348,179.234,6.105,149.325
C03252=1144.263,-45.364,-46.336,179.231,6.105,149.326
C03253=1144.268,-45.614,-46.325,179.229,6.104,149.326
C03254=1144.273,-45.864,-46.314,179.227,6.104,149.327
C03255=1144.279,-46.113,-46.303,179.225,6.103,149.328
C03256=1144.284,-46.363,-46.291,179.222,6.103,149.328
C03257=1144.289,-46.613,-46.280,179.220,6.102,149.329
C03258=1144.294,-46.862,-46.270,179.218,6.101,149.329
C03259=1144.300,-47.112,-46.258,179.215,6.101,149.330
C03260=1144.305,-47.362,-46.246,179.213,6.100,149.330
C03261=1144.310,-47.611,-46.236,179.211,6.099,149.331
C03262=1144.316,-47.861,-46.224,179.208,6.099,149.331
C03263=1144.320,-48.111,-46.213,179.206,6.098,149.332
C03264=1144.326,-48.361,-46.203,179.204,6.098,149.333
C03265=1144.331,-48.611,-46.191,179.201,6.098,149.333
C03266=1144.336,-48.860,-46.180,179.199,6.097,149.334
C03267=1144.342,-49.110,-46.170,179.197,6.096,149.334
C03268=1144.347,-49.360,-46.158,179.194,6.096,149.335
C03269=1144.352,-49.609,-46.147,179.192,6.095,149.335
C03270=1144.357,-49.859,-46.136,179.190,6.094,149.336
C03271=1144.363,-50.109,-46.124,179.187,6.094,149.337
C03272=1144.369,-50.379,-46.112,179.185,6.093,149.337
C03273=1144.374,-50.650,-46.101,179.182,6.093,149.338
C03274=1144.379,-50.921,-46.088,179.180,6.092,149.338
C03275=1144.386,-51.191,-46.077,179.178,6.092,149.339
C03276=1144.391,-51.441,-46.066,179.175,6.091,149.339
C03277=1144.395,-51.691,-46.055,179.173,6.090,149.340
C03278=1144.402,-51.941,-46.044,179.171,6.090,149.341
C03279=1144.406,-52.190,-46.033,179.169,6.090,149.341
C03280=1144.412,-52.440,-46.022,179.166,6.089,149.342
C03281=1144.417,-52.689,-46.011,179.164,6.089,149.342
C03282=1144.423,-52.939,-46.000,179.162,6.088,149.343
C03283=1144.428,-53.189,-45.989,179.159,6.087,149.344
C03284=1144.432,-53.439,-45.978,179.157,6.087,149.344
C03285=1144.438,-53.688,-45.968,179.155,6.087,149.344
C03286=1144.443,-53.938,-45.956,179.153,6.086,149.345
C03287=1144.449,-54.188,-45.945,179.151,6.085,149.346
C03288=1144.454,-54.437,-45.934,179.148,6.085,149.346
C03289=1144.459,-54.687,-45.924,179.146,6.084,149.347
C03290=1144.464,-54.937,-45.913,179.144,6.083,149.347
C03291=1144.470,-55.187,-45.901,179.141,6.083,149.348
C03292=1144.475,-55.436,-45.891,179.139,6.083,149.348
C03293=1144.480,-55.686,-45.880,179.137,6.082,149.349
C03294=1144.486,-55.936,-45.870,179.134,6.082,149.350
C03295=1144.490,-56.185,-45.858,179.132,6.081,149.350
C03296=1144.496,-56.435,-45.848,179.130,6.080,149.351
C03297=1144.501,-56.684,-45.837,179.127,6.080,149.351
C03298=1144.506,-56.935,-45.826,179.125,6.079,149.352
C03299=1144.512,-57.185,-45.816,179.124,6.079,149.352
C03300=1144.517,-57.434,-45.804,179.121,6.079,149.353
C03301=1144.522,-57.684,-45.794,179.119,6.078,149.353
C03302=1144.527,-57.933,-45.783,179.117,6.077,149.354
C03303=1144.533,-58.183,-45.773,179.114,6.077,149.355
C03304=1144.538,-58.433,-45.762,179.112,6.076,149.355
C03305=1144.543,-58.682,-45.751,179.110,6.076,149.356
C03306=1144.549,-58.933,-45.740,179.107,6.076,149.356
C03307=1144.554,-59.182,-45.730,179.105,6.075,149.357
C03308=1144.559,-59.432,-45.718,179.103,6.074,149.357
C03309=1144.564,-59.681,-45.708,179.100,6.074,149.358
C03310=1144.569,-59.932,-45.698,179.098,6.073,149.358
C03311=1144.575,-60.180,-45.687,179.097,6.073,149.359
C03312=1144.580,-60.431,-45.676,179.094,6.073,149.360
C03313=1144.585,-60.680,-45.666,179.092,6.072,149.360
C03314=1144.590,-60.930,-45.655,179.090,6.071,149.361
C03315=1144.596,-61.179,-45.644,179.087,6.071,149.361
C03316=1144.601,-61.430,-45.634,179.085,6.070,149.362
C03317=1144.606,-61.679,-45.624,179.083,6.070,149.362
C03318=1144.611,-61.929,-45.612,179.080,6.070,149.363
C03319=1144.617,-62.178,-45.602,179.078,6.069,149.363
C03320=1144.623,-62.428,-45.591,179.076,6.068,149.364
C03321=1144.628,-62.678,-45.581,179.073,6.068,149.365
C03322=1144.633,-62.927,-45.570,179.072,6.068,149.365
C03323=1144.638,-63.178,-45.559,179.070,6.067,149.366
C03324=1144.644,-63.427,-45.549,179.067,6.066,149.366
C03325=1144.649,-63.677,-45.538,179.065,6.066,149.367
C03326=1144.654,-63.926,-45.528,179.063,6.065,149.367
C03327=1144.659,-64.177,-45.517,179.061,6.065,149.368
C03328=1144.665,-64.426,-45.507,179.058,6.065,149.368
C03329=1144.670,-64.676,-45.497,179.056,6.064,149.369
C03330=1144.675,-64.926,-45.486,179.054,6.063,149.369
C03331=1144.681,-65.175,-45.476,179.051,6.063,149.370
C03332=1144.686,-65.425,-45.465,179.049,6.062,149.371
C03333=1144.690,-65.674,-45.455,179.047,6.062,149.371
C03334=1144.695,-65.925,-45.444,179.045,6.062,149.372
C03335=1144.701,-66.174,-45.434,179.043,6.061,149.372
C03336=1144.707,-66.424,-45.424,179.040,6.060,149.373
C03337=1144.712,-66.674,-45.413,179.038,6.060,149.373
C03338=1144.717,-66.923,-45.403,179.036,6.060,149.374
C03339=1144.722,-67.172,-45.392,179.034,6.059,149.374
C03340=1144.727,-67.423,-45.382,179.031,6.059,149.375
C03341=1144.733,-67.672,-45.371,179.029,6.058,149.376
C03342=1144.738,-67.922,-45.361,179.028,6.058,149.376
C03343=1144.744,-68.172,-45.351,179.025,6.057,149.377
C03344=1144.749,-68.422,-45.340,179.023,6.057,149.377
C03345=1144.754,-68.672,-45.330,179.020,6.056,149.378
C03346=1144.760,-68.921,-45.320,179.018,6.055,149.378
C03347=1144.765,-69.171,-45.309,179.016,6.055,149.379
C03348=1144.770,-69.421,-45.299,179.014,6.055,149.379
C03349=1144.775,-69.670,-45.289,179.012,6.054,149.380
C03350=1144.781,-69.920,-45.279,179.009,6.054,149.381
C03351=1144.786,-70.170,-45.268,179.008,6.054,149.381
C03352=1144.792,-70.420,-45.258,179.005,6.053,149.382
C03353=1144.797,-70.669,-45.248,179.003,6.052,149.382
C03354=1144.802,-70.919,-45.237,179.000,6.052,149.383
C03355=1144.808,-71.169,-45.227,178.998,6.051,149.383
C03356=1144.813,-71.418,-45.218,178.997,6.051,149.384
C03357=1144.818,-71.668,-45.207,178.994,6.051,149.384
C03358=1144.823,-71.918,-45.197,178.992,6.050,149.385
C03359=1144.829,-72.168,-45.187,178.990,6.049,149.385
C03360=1144.834,-72.418,-45.176,178.988,6.049,149.386
C03361=1144.839,-72.667,-45.166,178.985,6.049,149.387
C03362=1144.844,-72.917,-45.156,178.983,6.048,149.387
C03363=1144.849,-73.167,-45.146,178.981,6.047,149.388
C03364=1144.855,-73.416,-45.135,178.979,6.047,149.388
C03365=1144.860,-73.666,-45.125,178.977,6.047,149.389
C03366=1144.866,-73.915,-45.115,178.975,6.046,149.389
C03367=1144.871,-74.166,-45.104,178.972,6.046,149.390
C03368=1144.876,-74.415,-45.095,178.970,6.046,149.390
C03369=1144.882,-74.665,-45.085,178.968,6.045,149.391
C03370=1144.887,-74.915,-45.075,178.966,6.044,149.391
C03371=1144.892,-75.165,-45.065,178.963,6.044,149.392
C03372=1144.897,-75.414,-45.055,178.962,6.044,149.393
C03373=1144.903,-75.664,-45.045,178.959,6.043,149.393
C03374=1144.908,-75.914,-45.034,178.957,6.043,149.394
C03375=1144.913,-76.163,-45.024,178.955,6.042,149.394
C03376=1144.919,-76.435,-45.014,178.952,6.041,149.395
C03377=1144.925,-76.706,-45.003,178.950,6.041,149.395
C03378=1144.931,-76.978,-44.992,178.948,6.041,149.396
C03379=1144.937,-77.249,-44.980,178.945,6.040,149.397
C03380=1144.942,-77.499,-44.971,178.943,6.040,149.397
C03381=1144.947,-77.749,-44.961,178.941,6.039,149.398
C03382=1144.953,-77.998,-44.951,178.939,6.039,149.398
C03383=1144.958,-78.248,-44.940,178.937,6.038,149.399
C03384=1144.963,-78.498,-44.931,178.935,6.038,149.399
C03385=1144.969,-78.748,-44.921,178.932,6.037,149.400
C03386=1144.974,-78.997,-44.911,178.930,6.037,149.400
C03387=1144.979,-79.247,-44.901,178.928,6.037,149.401
C03388=1144.984,-79.497,-44.891,178.926,6.036,149.401
C03389=1144.990,-79.747,-44.881,178.924,6.036,149.402
C03390=1144.995,-79.996,-44.872,178.922,6.035,149.403
C03391=1145.001,-80.246,-44.861,178.919,6.035,149.403
C03392=1145.006,-80.496,-44.851,178.917,6.034,149.404
C03393=1145.011,-80.746,-44.842,178.915,6.034,149.404
C03394=1145.016,-80.995,-44.832,178.913,6.034,149.405
C03395=1145.022,-81.245,-44.822,178.911,6.033,149.405
C03396=1145.027,-81.495,-44.813,178.909,6.032,149.406
C03397=1145.033,-81.744,-44.802,178.907,6.032,149.406
C03398=1145.038,-81.995,-44.792,178.904,6.032,149.407
C03399=1145.043,-82.244,-44.783,178.902,6.031,149.407
C03400=1145.048,-82.494,-44.773,178.901,6.031,149.408
C03401=1145.054,-82.743,-44.763,178.898,6.031,149.409
C03402=1145.059,-82.993,-44.754,178.896,6.030,149.409
C03403=1145.065,-83.243,-44.743,178.894,6.030,149.410
C03404=1145.069,-83.493,-44.733,178.892,6.029,149.410
C03405=1145.075,-83.743,-44.724,178.889,6.029,149.411
C03406=1145.081,-83.992,-44.714,178.887,6.028,149.411
C03407=1145.085,-84.242,-44.704,178.885,6.028,149.412
C03408=1145.091,-84.492,-44.695,178.883,6.027,149.412
C03409=1145.096,-84.741,-44.685,178.881,6.027,149.413
C03410=1145.101,-84.991,-44.674,178.879,6.027,149.413
C03411=1145.106,-85.241,-44.666,178.877,6.026,149.414
C03412=1145.112,-85.491,-44.655,178.875,6.025,149.414
C03413=1145.118,-85.741,-44.646,178.873,6.026,149.415
C03414=1145.123,-85.990,-44.636,178.870,6.025,149.416
C03415=1145.129,-86.240,-44.627,178.868,6.024,149.416
C03416=1145.133,-86.490,-44.617,178.866,6.023,149.417
C03417=1145.138,-86.740,-44.607,178.864,6.024,149.417
C03418=1145.144,-86.990,-44.598,178.862,6.023,149.418
C03419=1145.149,-87.239,-44.587,178.860,6.022,149.418
C03420=1145.154,-87.489,-44.579,178.858,6.022,149.419
C03421=1145.160,-87.739,-44.568,178.855,6.022,149.419
C03422=1145.165,-87.988,-44.559,178.853,6.021,149.420
C03423=1145.171,-88.238,-44.549,178.851,6.021,149.420
C03424=1145.176,-88.488,-44.540,178.849,6.021,149.421
C03425=1145.181,-88.737,-44.530,178.847,6.020,149.422
C03426=1145.187,-88.987,-44.521,178.845,6.020,149.422
C03427=1145.192,-89.237,-44.511,178.843,6.019,149.423
C03428=1145.197,-89.487,-44.502,178.841,6.019,149.423
C03429=1145.202,-89.737,-44.492,178.839,6.019,149.424
C03430=1145.208,-89.987,-44.483,178.836,6.018,149.424
C03431=1145.213,-90.236,-44.472,178.834,6.018,149.425
C03432=1145.218,-90.486,-44.464,178.833,6.018,149.425
C03433=1145.224,-90.736,-44.453,178.830,6.017,149.426
C03434=1145.229,-90.985,-44.444,178.828,6.016,149.426
C03435=1145.235,-91.235,-44.434,178.826,6.017,149.427
C03436=1145.240,-91.485,-44.425,178.824,6.016,149.427
C03437=1145.245,-91.735,-44.416,178.822,6.015,149.428
C03438=1145.251,-91.984,-44.406,178.820,6.015,149.429
C03439=1145.256,-92.234,-44.397,178.817,6.015,149.429
C03440=1145.261,-92.484,-44.387,178.815,6.014,149.430
C03441=1145.267,-92.734,-44.378,178.814,6.014,149.430
C03442=1145.272,-92.984,-44.369,178.811,6.013,149.431
C03443=1145.277,-93.233,-44.359,178.809,6.013,149.431
C03444=1145.283,-93.483,-44.350,178.807,6.013,149.432
C03445=1145.288,-93.732,-44.340,178.805,6.012,149.432
C03446=1145.293,-93.983,-44.331,178.803,6.011,149.433
C03447=1145.299,-94.233,-44.321,178.801,6.011,149.433
C03448=1145.303,-94.482,-44.312,178.799,6.011,149.434
C03449=1145.309,-94.732,-44.303,178.796,6.010,149.434
C03450=1145.315,-94.982,-44.293,178.795,6.010,149.435
C03451=1145.319,-95.232,-44.284,178.793,6.009,149.435
C03452=1145.325,-95.482,-44.274,178.790,6.009,149.436
C03453=1145.330,-95.732,-44.265,178.788,6.009,149.437
C03454=1145.335,-95.981,-44.256,178.786,6.008,149.437
C03455=1145.341,-96.231,-44.246,178.784,6.008,149.438
C03456=1145.346,-96.481,-44.237,178.782,6.008,149.438
C03457=1145.352,-96.730,-44.229,178.780,6.007,149.438
C03458=1145.358,-96.979,-44.218,178.778,6.007,149.439
C03459=1145.363,-97.229,-44.210,178.776,6.007,149.440
C03460=1145.368,-97.479,-44.201,178.774,6.006,149.440
C03461=1145.374,-97.729,-44.190,178.772,6.006,149.441
C03462=1145.379,-97.979,-44.182,178.770,6.005,149.441
C03463=1145.384,-98.228,-44.173,178.767,6.005,149.442
C03464=1145.390,-98.479,-44.163,178.766,6.005,149.442
C03465=1145.395,-98.728,-44.154,178.763,6.004,149.443
C03466=1145.400,-98.978,-44.145,178.761,6.003,149.443
C03467=1145.406,-99.228,-44.135,178.760,6.003,149.444
C03468=1145.411,-99.478,-44.126,178.757,6.003,149.444
C03469=1145.416,-99.728,-44.117,178.755,6.003,149.445
C03470=1145.421,-99.977,-44.108,178.753,6.002,149.445
C03471=1145.427,-100.227,-44.098,178.751,6.001,149.446
C03472=1145.432,-100.477,-44.089,178.749,6.001,149.446
C03473=1145.437,-100.727,-44.080,178.747,6.001,149.447
C03474=1145.443,-100.977,-44.071,178.744,6.000,149.448
C03475=1145.448,-101.227,-44.062,178.743,6.000,149.448
C03476=1145.453,-101.476,-44.052,178.741,6.000,149.449
C03477=1145.459,-101.725,-44.044,178.739,6.000,149.449
C03478=1145.465,-101.975,-44.034,178.737,5.999,149.450
C03479=1145.470,-102.225,-44.026,178.734,5.999,149.450
C03480=1145.476,-102.497,-44.015,178.733,5.999,149.451
C03481=1145.481,-102.770,-44.006,178.730,5.998,149.451
C03482=1145.487,-103.041,-43.996,178.728,5.998,149.452
C03483=1145.493,-103.314,-43.986,178.726,5.997,149.452
C03484=1145.498,-103.564,-43.977,178.724,5.997,149.453
C03485=1145.504,-103.813,-43.968,178.722,5.996,149.453
C03486=1145.509,-104.063,-43.958,178.720,5.996,149.454
C03487=1145.514,-104.312,-43.950,178.717,5.996,149.455
C03488=1145.519,-104.562,-43.941,178.715,5.995,149.455
C03489=1145.525,-104.812,-43.932,178.714,5.995,149.456
C03490=1145.531,-105.062,-43.922,178.711,5.994,149.456
C03491=1145.536,-105.312,-43.913,178.710,5.994,149.457
C03492=1145.541,-105.562,-43.904,178.708,5.994,149.457
C03493=1145.546,-105.812,-43.896,178.705,5.993,149.458
C03494=1145.552,-106.061,-43.887,178.703,5.993,149.458
C03495=1145.557,-106.311,-43.878,178.701,5.992,149.459
C03496=1145.563,-106.561,-43.869,178.700,5.992,149.459
C03497=1145.568,-106.811,-43.860,178.697,5.992,149.460
C03498=1145.573,-107.061,-43.851,178.695,5.991,149.460
C03499=1145.578,-107.311,-43.842,178.693,5.991,149.461
C03500=1145.584,-107.560,-43.833,178.691,5.991,149.461
C03501=1145.589,-107.810,-43.825,178.689,5.991,149.462
C03502=1145.594,-108.059,-43.816,178.687,5.990,149.462
C03503=1145.600,-108.310,-43.806,178.685,5.989,149.463
C03504=1145.606,-108.559,-43.797,178.683,5.989,149.463
C03505=1145.611,-108.809,-43.788,178.681,5.988,149.464
C03506=1145.616,-109.059,-43.779,178.679,5.989,149.465
C03507=1145.622,-109.308,-43.771,178.677,5.988,149.465
C03508=1145.627,-109.558,-43.762,178.675,5.988,149.466
C03509=1145.632,-109.808,-43.753,178.673,5.987,149.466
C03510=1145.637,-110.058,-43.744,178.671,5.987,149.467
C03511=1145.642,-110.308,-43.735,178.669,5.987,149.467
C03512=1145.648,-110.557,-43.727,178.667,5.986,149.467
C03513=1145.654,-110.807,-43.717,178.665,5.986,149.468
C03514=1145.659,-111.057,-43.708,178.663,5.986,149.469
C03515=1145.664,-111.307,-43.699,178.661,5.985,149.469
C03516=1145.670,-111.557,-43.691,178.659,5.985,149.470
C03517=1145.676,-111.806,-43.683,178.657,5.984,149.470
C03518=1145.681,-112.056,-43.674,178.655,5.984,149.471
C03519=1145.686,-112.306,-43.665,178.653,5.983,149.471
C03520=1145.691,-112.556,-43.656,178.651,5.983,149.472
C03521=1145.697,-112.805,-43.648,178.649,5.983,149.472
C03522=1145.702,-113.055,-43.639,178.647,5.982,149.473
C03523=1145.707,-113.305,-43.630,178.645,5.982,149.473
C03524=1145.713,-113.555,-43.622,178.643,5.982,149.474
C03525=1145.718,-113.805,-43.613,178.641,5.982,149.474
C03526=1145.724,-114.054,-43.604,178.639,5.981,149.475
C03527=1145.729,-114.304,-43.595,178.637,5.981,149.475
C03528=1145.734,-114.554,-43.586,178.635,5.980,149.476
C03529=1145.739,-114.804,-43.577,178.634,5.980,149.476
C03530=1145.745,-115.053,-43.570,178.631,5.980,149.477
C03531=1145.750,-115.303,-43.561,178.629,5.979,149.477
C03532=1145.755,-115.553,-43.552,178.627,5.979,149.478
C03533=1145.761,-115.803,-43.543,178.625,5.978,149.478
C03534=1145.766,-116.052,-43.534,178.623,5.979,149.479
C03535=1145.772,-116.303,-43.526,178.621,5.978,149.479
C03536=1145.777,-116.552,-43.517,178.620,5.978,149.480
C03537=1145.783,-116.802,-43.509,178.617,5.977,149.480
C03538=1145.788,-117.051,-43.500,178.616,5.977,149.481
C03539=1145.793,-117.302,-43.492,178.614,5.976,149.481
C03540=1145.799,-117.552,-43.483,178.611,5.976,149.482
C03541=1145.804,-117.801,-43.474,178.609,5.976,149.482
C03542=1145.810,-118.051,-43.465,178.607,5.975,149.483
C03543=1145.815,-118.301,-43.457,178.605,5.975,149.483
C03544=1145.821,-118.550,-43.449,178.603,5.975,149.484
C03545=1145.826,-118.800,-43.440,178.602,5.975,149.484
C03546=1145.831,-119.050,-43.431,178.599,5.974,149.485
C03547=1145.837,-119.301,-43.423,178.598,5.974,149.485
C03548=1145.842,-119.550,-43.414,178.596,5.973,149.486
C03549=1145.847,-119.799,-43.406,178.594,5.973,149.486
C03550=1145.852,-120.050,-43.398,178.592,5.972,149.487
C03551=1145.858,-120.299,-43.389,178.590,5.973,149.488
C03552=1145.863,-120.549,-43.380,178.588,5.972,149.488
C03553=1145.869,-120.799,-43.372,178.586,5.972,149.489
C03554=1145.874,-121.048,-43.364,178.584,5.971,149.489
C03555=1145.880,-121.298,-43.355,178.582,5.971,149.490
C03556=1145.885,-121.549,-43.346,178.580,5.971,149.490
C03557=1145.891,-121.798,-43.338,178.578,5.970,149.491
C03558=1145.895,-122.047,-43.330,178.576,5.970,149.491
C03559=1145.901,-122.298,-43.321,178.574,5.969,149.492
C03560=1145.907,-122.547,-43.313,178.572,5.969,149.492
C03561=1145.912,-122.797,-43.304,178.570,5.969,149.492
C03562=1145.917,-123.047,-43.296,178.569,5.969,149.493
C03563=1145.923,-123.296,-43.287,178.566,5.968,149.493
C03564=1145.928,-123.547,-43.279,178.565,5.968,149.494
C03565=1145.933,-123.796,-43.271,178.562,5.968,149.495
C03566=1145.939,-124.046,-43.262,178.561,5.968,149.495
C03567=1145.944,-124.296,-43.254,178.558,5.967,149.496
C03568=1145.950,-124.545,-43.246,178.557,5.967,149.496
C03569=1145.955,-124.796,-43.237,178.555,5.966,149.497
C03570=1145.960,-125.046,-43.228,178.553,5.966,149.497
C03571=1145.966,-125.295,-43.221,178.551,5.965,149.498
C03572=1145.971,-125.545,-43.212,178.549,5.965,149.498
C03573=1145.976,-125.795,-43.204,178.547,5.965,149.499
C03574=1145.982,-126.045,-43.196,178.545,5.965,149.499
C03575=1145.987,-126.294,-43.187,178.543,5.964,149.500
C03576=1145.993,-126.544,-43.180,178.542,5.964,149.500
C03577=1145.998,-126.794,-43.171,178.539,5.963,149.501
C03578=1146.003,-127.044,-43.162,178.538,5.963,149.501
C03579=1146.009,-127.293,-43.154,178.536,5.963,149.501
C03580=1146.015,-127.544,-43.146,178.534,5.963,149.502
C03581=1146.020,-127.793,-43.138,178.532,5.962,149.502
C03582=1146.025,-128.043,-43.130,178.530,5.962,149.503
C03583=1146.030,-128.293,-43.121,178.528,5.961,149.503
C03584=1145.610,-128.304,-43.164,178.524,5.965,149.505
C03585=1145.604,-128.054,-43.172,178.526,5.965,149.505
C03586=1145.599,-127.805,-43.181,178.528,5.965,149.504
C03587=1145.593,-127.554,-43.189,178.530,5.966,149.504
C03588=1145.588,-127.305,-43.197,178.532,5.967,149.503
C03589=1145.583,-127.055,-43.205,178.534,5.967,149.503
C03590=1145.578,-126.805,-43.214,178.536,5.967,149.502
C03591=1145.571,-126.555,-43.222,178.538,5.967,149.502
C03592=1145.566,-126.305,-43.231,178.540,5.968,149.501
C03593=1145.561,-126.056,-43.238,178.542,5.968,149.501
C03594=1145.556,-125.806,-43.247,178.544,5.969,149.500
C03595=1145.550,-125.556,-43.255,178.545,5.969,149.500
C03596=1145.545,-125.307,-43.264,178.548,5.970,149.499
C03597=1145.539,-125.056,-43.272,178.549,5.969,149.499
C03598=1145.534,-124.807,-43.280,178.551,5.970,149.498
C03599=1145.529,-124.557,-43.289,178.553,5.970,149.498
C03600=1145.523,-124.307,-43.297,178.556,5.971,149.497
C03601=1145.518,-124.058,-43.305,178.557,5.970,149.497
C03602=1145.512,-123.807,-43.314,178.559,5.971,149.496
C03603=1145.507,-123.557,-43.323,178.561,5.971,149.496
C03604=1145.502,-123.308,-43.330,178.563,5.972,149.495
C03605=1145.497,-123.058,-43.339,178.565,5.972,149.495
C03606=1145.491,-122.808,-43.348,178.567,5.973,149.494
C03607=1145.485,-122.559,-43.355,178.569,5.973,149.494
C03608=1145.480,-122.309,-43.364,178.571,5.973,149.493
C03609=1145.475,-122.059,-43.373,178.572,5.973,149.493
C03610=1145.469,-121.809,-43.381,178.575,5.974,149.492
C03611=1145.464,-121.560,-43.389,178.576,5.974,149.492
C03612=1145.459,-121.310,-43.398,178.578,5.975,149.491
C03613=1145.453,-121.060,-43.406,178.580,5.975,149.491
C03614=1145.448,-120.810,-43.415,178.582,5.975,149.490
C03615=1145.443,-120.560,-43.423,178.584,5.975,149.490
C03616=1145.437,-120.310,-43.432,178.586,5.976,149.489
C03617=1145.432,-120.061,-43.440,178.589,5.977,149.489
C03618=1145.426,-119.811,-43.449,178.590,5.976,149.488
C03619=1145.420,-119.561,-43.457,178.592,5.977,149.488
C03620=1145.415,-119.311,-43.466,178.594,5.977,149.487
C03621=1145.411,-119.062,-43.474,178.596,5.978,149.487
C03622=1145.405,-118.812,-43.482,178.598,5.978,149.486
C03623=1145.400,-118.562,-43.491,178.600,5.979,149.486
C03624=1145.394,-118.312,-43.500,178.602,5.979,149.485
C03625=1145.389,-118.062,-43.508,178.604,5.979,149.485
C03626=1145.383,-117.812,-43.517,178.605,5.979,149.484
C03627=1145.378,-117.563,-43.526,178.608,5.980,149.484
C03628=1145.373,-117.313,-43.535,178.610,5.980,149.483
C03629=1145.367,-117.063,-43.542,178.612,5.980,149.483
C03630=1145.362,-116.813,-43.551,178.614,5.981,149.482
C03631=1145.356,-116.563,-43.560,178.616,5.981,149.482
C03632=1145.351,-116.313,-43.569,178.618,5.982,149.481
C03633=1145.345,-116.064,-43.578,178.619,5.982,149.481
C03634=1145.340,-115.814,-43.586,178.622,5.983,149.480
C03635=1145.335,-115.564,-43.595,178.623,5.982,149.480
C03636=1145.329,-115.315,-43.603,178.625,5.983,149.479
